gfCNCPoint6[9679] = {X 429.6854, Y 18.4377, Z -8.0000, A 0.000, B 0.000, C 0.000 }
gfCNCPoint6[9680] = {X 430.1103, Y 16.6184, Z -8.0000, A 0.000, B 0.000, C 0.000 }
gfCNCPoint6[9681] = {X 430.6685, Y 15.1182, Z -8.0000, A 0.000, B 0.000, C 0.000 }
gfCNCPoint6[9682] = {X 431.4282, Y 13.7093, Z -8.0000, A 0.000, B 0.000, C 0.000 }
gfCNCPoint6[9683] = {X 432.3747, Y 12.4184, Z -8.0000, A 0.000, B 0.000, C 0.000 }
gfCNCPoint6[9684] = {X 433.4901, Y 11.2703, Z -8.0000, A 0.000, B 0.000, C 0.000 }
gfCNCPoint6[9685] = {X 434.7530, Y 10.2868, Z -8.0000, A 0.000, B 0.000, C 0.000 }
gfCNCPoint6[9686] = {X 436.1394, Y 9.4867, Z -8.0000, A 0.000, B 0.000, C 0.000 }
gfCNCPoint6[9687] = {X 437.6228, Y 8.8852, Z -8.0000, A 0.000, B 0.000, C 0.000 }
gfCNCPoint6[9688] = {X 439.1749, Y 8.4939, Z -8.0000, A 0.000, B 0.000, C 0.000 }
gfCNCPoint6[9689] = {X 441.2506, Y 8.2065, Z -8.0000, A 0.000, B 0.000, C 0.000 }
gfCNCPoint6[9690] = {X 443.3440, Y 8.1133, Z -8.0000, A 0.000, B 0.000, C 0.000 }
gfCNCPoint6[9691] = {X 444.0364, Y 8.1092, Z -8.0000, A 0.000, B 0.000, C 0.000 }
gfCNCPoint6[9692] = {X 459.4469, Y 8.1092, Z -8.0000, A 0.000, B 0.000, C 0.000 }
gfCNCPoint6[9693] = {X 460.3528, Y 8.2113, Z -8.0000, A 0.000, B 0.000, C 0.000 }
gfCNCPoint6[9694] = {X 461.2133, Y 8.5124, Z -8.0000, A 0.000, B 0.000, C 0.000 }
gfCNCPoint6[9695] = {X 461.9852, Y 8.9974, Z -8.0000, A 0.000, B 0.000, C 0.000 }
gfCNCPoint6[9696] = {X 462.6298, Y 9.6420, Z -8.0000, A 0.000, B 0.000, C 0.000 }
gfCNCPoint6[9697] = {X 463.1148, Y 10.4139, Z -8.0000, A 0.000, B 0.000, C 0.000 }
gfCNCPoint6[9698] = {X 463.4159, Y 11.2744, Z -8.0000, A 0.000, B 0.000, C 0.000 }
gfCNCPoint6[9699] = {X 463.5179, Y 12.1803, Z -8.0000, A 0.000, B 0.000, C 0.000 }
gfCNCPoint6[9700] = {X 463.5179, Y 12.9782, Z -8.0000, A 0.000, B 0.000, C 0.000 }
gfCNCPoint6[9701] = {X 463.4242, Y 13.8477, Z -8.0000, A 0.000, B 0.000, C 0.000 }
gfCNCPoint6[9702] = {X 463.1473, Y 14.6772, Z -8.0000, A 0.000, B 0.000, C 0.000 }
gfCNCPoint6[9703] = {X 462.6999, Y 15.4287, Z -8.0000, A 0.000, B 0.000, C 0.000 }
gfCNCPoint6[9704] = {X 462.1027, Y 16.0676, Z -8.0000, A 0.000, B 0.000, C 0.000 }
gfCNCPoint6[9705] = {X 462.0451, Y 16.1164, Z -8.0000, A 0.000, B 0.000, C 0.000 }
gfCNCPoint6[9706] = {X 461.9865, Y 16.1641, Z -8.0000, A 0.000, B 0.000, C 0.000 }
gfCNCPoint6[9707] = {X 461.9918, Y 16.1980, Z -8.0000, A 0.000, B 0.000, C 0.000 }
gfCNCPoint6[9708] = {X 461.9920, Y 28.5935, Z -8.0000, A 0.000, B 0.000, C 0.000 }
gfCNCPoint6[9709] = {X 465.9920, Y 28.5934, Z -8.0000, A 0.000, B 0.000, C 0.000 }
gfCNCPoint6[9710] = {X 465.9920, Y 28.5933, Z -8.0000, A 0.000, B 0.000, C 0.000 }
gfCNCPoint6[9711] = {X 461.9118, Y 28.5935, Z -8.0000, A 0.000, B 0.000, C 0.000 }
gfCNCPoint6[9712] = {X 461.9123, Y 41.0648, Z -8.0000, A 0.000, B 0.000, C 0.000 }
gfCNCPoint6[9713] = {X 462.0510, Y 41.1802, Z -8.0000, A 0.000, B 0.000, C 0.000 }
gfCNCPoint6[9714] = {X 462.6363, Y 41.8066, Z -8.0000, A 0.000, B 0.000, C 0.000 }
gfCNCPoint6[9715] = {X 463.0747, Y 42.5433, Z -8.0000, A 0.000, B 0.000, C 0.000 }
gfCNCPoint6[9716] = {X 463.3461, Y 43.3565, Z -8.0000, A 0.000, B 0.000, C 0.000 }
gfCNCPoint6[9717] = {X 463.4379, Y 44.2088, Z -8.0000, A 0.000, B 0.000, C 0.000 }
gfCNCPoint6[9718] = {X 463.4379, Y 45.0000, Z -8.0000, A 0.000, B 0.000, C 0.000 }
gfCNCPoint6[9719] = {X 463.3377, Y 45.8901, Z -8.0000, A 0.000, B 0.000, C 0.000 }
gfCNCPoint6[9720] = {X 463.0418, Y 46.7355, Z -8.0000, A 0.000, B 0.000, C 0.000 }
gfCNCPoint6[9721] = {X 462.5653, Y 47.4940, Z -8.0000, A 0.000, B 0.000, C 0.000 }
gfCNCPoint6[9722] = {X 461.9319, Y 48.1273, Z -8.0000, A 0.000, B 0.000, C 0.000 }
gfCNCPoint6[9723] = {X 461.1735, Y 48.6039, Z -8.0000, A 0.000, B 0.000, C 0.000 }
gfCNCPoint6[9724] = {X 460.3280, Y 48.8997, Z -8.0000, A 0.000, B 0.000, C 0.000 }
gfCNCPoint6[9725] = {X 459.4379, Y 49.0000, Z -8.0000, A 0.000, B 0.000, C 0.000 }
gfCNCPoint6[9726] = {X 452.9945, Y 49.0000, Z -8.0000, A 0.000, B 0.000, C 0.000 }
gfCNCPoint6[9727] = {X 452.1044, Y 48.8997, Z -8.0000, A 0.000, B 0.000, C 0.000 }
gfCNCPoint6[9728] = {X 451.2589, Y 48.6039, Z -8.0000, A 0.000, B 0.000, C 0.000 }
gfCNCPoint6[9729] = {X 450.5005, Y 48.1273, Z -8.0000, A 0.000, B 0.000, C 0.000 }
gfCNCPoint6[9730] = {X 449.8671, Y 47.4939, Z -8.0000, A 0.000, B 0.000, C 0.000 }
gfCNCPoint6[9731] = {X 449.3906, Y 46.7355, Z -8.0000, A 0.000, B 0.000, C 0.000 }
gfCNCPoint6[9732] = {X 449.0948, Y 45.8901, Z -8.0000, A 0.000, B 0.000, C 0.000 }
gfCNCPoint6[9733] = {X 448.9945, Y 45.0000, Z -8.0000, A 0.000, B 0.000, C 0.000 }
gfCNCPoint6[9734] = {X 448.9949, Y 44.1538, Z -8.0000, A 0.000, B 0.000, C 0.000 }
gfCNCPoint6[9735] = {X 449.1055, Y 43.2730, Z -8.0000, A 0.000, B 0.000, C 0.000 }
gfCNCPoint6[9736] = {X 449.4077, Y 42.4382, Z -8.0000, A 0.000, B 0.000, C 0.000 }
gfCNCPoint6[9737] = {X 449.8865, Y 41.6907, Z -8.0000, A 0.000, B 0.000, C 0.000 }
gfCNCPoint6[9738] = {X 450.5184, Y 41.0672, Z -8.0000, A 0.000, B 0.000, C 0.000 }
gfCNCPoint6[9739] = {X 450.5184, Y 34.1538, Z -8.0000, A 0.000, B 0.000, C 0.000 }
gfCNCPoint6[9740] = {X 447.2803, Y 34.1538, Z -8.0000, A 0.000, B 0.000, C 0.000 }
gfCNCPoint6[9741] = {X 442.8423, Y 42.7952, Z -8.0000, A 0.000, B 0.000, C 0.000 }
gfCNCPoint6[9742] = {X 442.8973, Y 42.9503, Z -8.0000, A 0.000, B 0.000, C 0.000 }
gfCNCPoint6[9743] = {X 443.0494, Y 43.5714, Z -8.0000, A 0.000, B 0.000, C 0.000 }
gfCNCPoint6[9744] = {X 443.1005, Y 44.2089, Z -8.0000, A 0.000, B 0.000, C 0.000 }
gfCNCPoint6[9745] = {X 443.1005, Y 45.0000, Z -8.0000, A 0.000, B 0.000, C 0.000 }
gfCNCPoint6[9746] = {X 443.0002, Y 45.8901, Z -8.0000, A 0.000, B 0.000, C 0.000 }
gfCNCPoint6[9747] = {X 442.7043, Y 46.7355, Z -8.0000, A 0.000, B 0.000, C 0.000 }
gfCNCPoint6[9748] = {X 442.2278, Y 47.4940, Z -8.0000, A 0.000, B 0.000, C 0.000 }
gfCNCPoint6[9749] = {X 441.5944, Y 48.1273, Z -8.0000, A 0.000, B 0.000, C 0.000 }
gfCNCPoint6[9750] = {X 440.8360, Y 48.6039, Z -8.0000, A 0.000, B 0.000, C 0.000 }
gfCNCPoint6[9751] = {X 439.9906, Y 48.8997, Z -8.0000, A 0.000, B 0.000, C 0.000 }
gfCNCPoint6[9752] = {X 439.1005, Y 49.0000, Z -8.0000, A 0.000, B 0.000, C 0.000 }
gfCNCPoint6[9753] = {X 432.5144, Y 49.0000, Z -8.0000, A 0.000, B 0.000, C 0.000 }
gfCNCPoint6[9754] = {X 431.6243, Y 48.8997, Z -8.0000, A 0.000, B 0.000, C 0.000 }
gfCNCPoint6[9755] = {X 430.7789, Y 48.6039, Z -8.0000, A 0.000, B 0.000, C 0.000 }
gfCNCPoint6[9756] = {X 430.0204, Y 48.1273, Z -8.0000, A 0.000, B 0.000, C 0.000 }
gfCNCPoint6[9757] = {X 429.3871, Y 47.4940, Z -8.0000, A 0.000, B 0.000, C 0.000 }
gfCNCPoint6[9758] = {X 428.9105, Y 46.7355, Z -8.0000, A 0.000, B 0.000, C 0.000 }
gfCNCPoint6[9759] = {X 428.6147, Y 45.8901, Z -8.0000, A 0.000, B 0.000, C 0.000 }
gfCNCPoint6[9760] = {X 428.5144, Y 45.0000, Z -8.0000, A 0.000, B 0.000, C 0.000 }
gfCNCPoint6[9761] = {X 428.5148, Y 44.1538, Z -8.0000, A 0.000, B 0.000, C 0.000 }
gfCNCPoint6[9762] = {X 428.6096, Y 43.3414, Z -8.0000, A 0.000, B 0.000, C 0.000 }
gfCNCPoint6[9763] = {X 428.8676, Y 42.5654, Z -8.0000, A 0.000, B 0.000, C 0.000 }
gfCNCPoint6[9764] = {X 429.2781, Y 41.8580, Z -8.0000, A 0.000, B 0.000, C 0.000 }
gfCNCPoint6[9765] = {X 429.8239, Y 41.2489, Z -8.0000, A 0.000, B 0.000, C 0.000 }
gfCNCPoint6[9766] = {X 430.4821, Y 40.7635, Z -8.0000, A 0.000, B 0.000, C 0.000 }
gfCNCPoint6[9767] = {X 431.2253, Y 40.4222, Z -8.0000, A 0.000, B 0.000, C 0.000 }
gfCNCPoint6[9768] = {X 435.4110, Y 32.2292, Z -8.0000, A 0.000, B 0.000, C 0.000 }
gfCNCPoint6[9769] = {X 434.2190, Y 31.4711, Z -8.0000, A 0.000, B 0.000, C 0.000 }
gfCNCPoint6[9770] = {X 433.1339, Y 30.5665, Z -8.0000, A 0.000, B 0.000, C 0.000 }
gfCNCPoint6[9771] = {X 432.1736, Y 29.5306, Z -8.0000, A 0.000, B 0.000, C 0.000 }
gfCNCPoint6[9772] = {X 431.3537, Y 28.3802, Z -8.0000, A 0.000, B 0.000, C 0.000 }
gfCNCPoint6[9773] = {X 430.6879, Y 27.1343, Z -8.0000, A 0.000, B 0.000, C 0.000 }
gfCNCPoint6[9774] = {X 430.1870, Y 25.8134, Z -8.0000, A 0.000, B 0.000, C 0.000 }
gfCNCPoint6[9775] = {X 429.7643, Y 24.0033, Z -8.0000, A 0.000, B 0.000, C 0.000 }
gfCNCPoint6[9776] = {X 429.5515, Y 22.1566, Z -8.0000, A 0.000, B 0.000, C 0.000 }
gfCNCPoint6[9777] = {X 429.5515, Y 20.2978, Z -8.0000, A 0.000, B 0.000, C 0.000 }
gfCNCPoint6[9778] = {X 429.7643, Y 18.4512, Z -8.0000, A 0.000, B 0.000, C 0.000 }
gfCNCPoint6[9779] = {X 430.1870, Y 16.6411, Z -8.0000, A 0.000, B 0.000, C 0.000 }
gfCNCPoint6[9780] = {X 430.7414, Y 15.1512, Z -8.0000, A 0.000, B 0.000, C 0.000 }
gfCNCPoint6[9781] = {X 431.4958, Y 13.7519, Z -8.0000, A 0.000, B 0.000, C 0.000 }
gfCNCPoint6[9782] = {X 432.4359, Y 12.4700, Z -8.0000, A 0.000, B 0.000, C 0.000 }
gfCNCPoint6[9783] = {X 433.5436, Y 11.3298, Z -8.0000, A 0.000, B 0.000, C 0.000 }
gfCNCPoint6[9784] = {X 434.7978, Y 10.3531, Z -8.0000, A 0.000, B 0.000, C 0.000 }
gfCNCPoint6[9785] = {X 436.1746, Y 9.5585, Z -8.0000, A 0.000, B 0.000, C 0.000 }
gfCNCPoint6[9786] = {X 437.6478, Y 8.9612, Z -8.0000, A 0.000, B 0.000, C 0.000 }
gfCNCPoint6[9787] = {X 439.1893, Y 8.5726, Z -8.0000, A 0.000, B 0.000, C 0.000 }
gfCNCPoint6[9788] = {X 441.2579, Y 8.2861, Z -8.0000, A 0.000, B 0.000, C 0.000 }
gfCNCPoint6[9789] = {X 443.3442, Y 8.1933, Z -8.0000, A 0.000, B 0.000, C 0.000 }
gfCNCPoint6[9790] = {X 444.0367, Y 8.1892, Z -8.0000, A 0.000, B 0.000, C 0.000 }
gfCNCPoint6[9791] = {X 459.4469, Y 8.1892, Z -8.0000, A 0.000, B 0.000, C 0.000 }
gfCNCPoint6[9792] = {X 460.3350, Y 8.2893, Z -8.0000, A 0.000, B 0.000, C 0.000 }
gfCNCPoint6[9793] = {X 461.1786, Y 8.5845, Z -8.0000, A 0.000, B 0.000, C 0.000 }
gfCNCPoint6[9794] = {X 461.9353, Y 9.0600, Z -8.0000, A 0.000, B 0.000, C 0.000 }
gfCNCPoint6[9795] = {X 462.5672, Y 9.6919, Z -8.0000, A 0.000, B 0.000, C 0.000 }
gfCNCPoint6[9796] = {X 463.0427, Y 10.4486, Z -8.0000, A 0.000, B 0.000, C 0.000 }
gfCNCPoint6[9797] = {X 463.3379, Y 11.2922, Z -8.0000, A 0.000, B 0.000, C 0.000 }
gfCNCPoint6[9798] = {X 463.4379, Y 12.1803, Z -8.0000, A 0.000, B 0.000, C 0.000 }
gfCNCPoint6[9799] = {X 463.4378, Y 13.0163, Z -8.0000, A 0.000, B 0.000, C 0.000 }
gfCNCPoint6[9800] = {X 463.3398, Y 13.8585, Z -8.0000, A 0.000, B 0.000, C 0.000 }
gfCNCPoint6[9801] = {X 463.0666, Y 14.6612, Z -8.0000, A 0.000, B 0.000, C 0.000 }
gfCNCPoint6[9802] = {X 462.6302, Y 15.3883, Z -8.0000, A 0.000, B 0.000, C 0.000 }
gfCNCPoint6[9803] = {X 462.0505, Y 16.0070, Z -8.0000, A 0.000, B 0.000, C 0.000 }
gfCNCPoint6[9804] = {X 461.9731, Y 16.0720, Z -8.0000, A 0.000, B 0.000, C 0.000 }
gfCNCPoint6[9805] = {X 461.8942, Y 16.1351, Z -8.0000, A 0.000, B 0.000, C 0.000 }
gfCNCPoint6[9806] = {X 461.9118, Y 16.1935, Z -8.0000, A 0.000, B 0.000, C 0.000 }
gfCNCPoint6[9807] = {X 461.9113, Y 16.7687, Z -8.0000, A 0.000, B 0.000, C 0.000 }
gfCNCPoint6[9808] = {X 461.9118, Y 28.5935, Z -8.0000, A 0.000, B 0.000, C 0.000 }
gfCNCPoint6[9809] = {X 465.9920, Y 28.5933, Z -8.0000, A 0.000, B 0.000, C 0.000 }
gfCNCPoint6[9810] = {X 465.9920, Y 28.5933, Z -5.0000, A 0.000, B 0.000, C 0.000 }
gfCNCPoint6[9811] = {X 465.9920, Y 28.5933, Z 11.0000, A 0.000, B 0.000, C 0.000 }
gfCNCPoint6[9812] = {X 492.3835, Y 3.7892, Z 11.0000, A 0.000, B 0.000, C 0.000 }
gfCNCPoint6[9813] = {X 492.3835, Y 3.7892, Z -5.0000, A 0.000, B 0.000, C 0.000 }
gfCNCPoint6[9814] = {X 492.3835, Y 3.7892, Z -8.0000, A 0.000, B 0.000, C 0.000 }
gfCNCPoint6[9815] = {X 492.3835, Y 7.8692, Z -8.0000, A 0.000, B 0.000, C 0.000 }
gfCNCPoint6[9816] = {X 502.2066, Y 7.8692, Z -8.0000, A 0.000, B 0.000, C 0.000 }
gfCNCPoint6[9817] = {X 502.7394, Y 7.8734, Z -8.0000, A 0.000, B 0.000, C 0.000 }
gfCNCPoint6[9818] = {X 503.6913, Y 7.9876, Z -8.0000, A 0.000, B 0.000, C 0.000 }
gfCNCPoint6[9819] = {X 504.5943, Y 8.3098, Z -8.0000, A 0.000, B 0.000, C 0.000 }
gfCNCPoint6[9820] = {X 505.4035, Y 8.8240, Z -8.0000, A 0.000, B 0.000, C 0.000 }
gfCNCPoint6[9821] = {X 506.0787, Y 9.5045, Z -8.0000, A 0.000, B 0.000, C 0.000 }
gfCNCPoint6[9822] = {X 506.5865, Y 10.3177, Z -8.0000, A 0.000, B 0.000, C 0.000 }
gfCNCPoint6[9823] = {X 506.9017, Y 11.2232, Z -8.0000, A 0.000, B 0.000, C 0.000 }
gfCNCPoint6[9824] = {X 507.0085, Y 12.1759, Z -8.0000, A 0.000, B 0.000, C 0.000 }
gfCNCPoint6[9825] = {X 507.0085, Y 12.9782, Z -8.0000, A 0.000, B 0.000, C 0.000 }
gfCNCPoint6[9826] = {X 506.9072, Y 13.9079, Z -8.0000, A 0.000, B 0.000, C 0.000 }
gfCNCPoint6[9827] = {X 506.6082, Y 14.7940, Z -8.0000, A 0.000, B 0.000, C 0.000 }
gfCNCPoint6[9828] = {X 506.1256, Y 15.5951, Z -8.0000, A 0.000, B 0.000, C 0.000 }
gfCNCPoint6[9829] = {X 505.4818, Y 16.2734, Z -8.0000, A 0.000, B 0.000, C 0.000 }
gfCNCPoint6[9830] = {X 505.4824, Y 40.9138, Z -8.0000, A 0.000, B 0.000, C 0.000 }
gfCNCPoint6[9831] = {X 506.1202, Y 41.5848, Z -8.0000, A 0.000, B 0.000, C 0.000 }
gfCNCPoint6[9832] = {X 506.6005, Y 42.3762, Z -8.0000, A 0.000, B 0.000, C 0.000 }
gfCNCPoint6[9833] = {X 506.9012, Y 43.2518, Z -8.0000, A 0.000, B 0.000, C 0.000 }
gfCNCPoint6[9834] = {X 507.0083, Y 44.1713, Z -8.0000, A 0.000, B 0.000, C 0.000 }
gfCNCPoint6[9835] = {X 507.0085, Y 45.0000, Z -8.0000, A 0.000, B 0.000, C 0.000 }
gfCNCPoint6[9836] = {X 506.9002, Y 45.9613, Z -8.0000, A 0.000, B 0.000, C 0.000 }
gfCNCPoint6[9837] = {X 506.5807, Y 46.8744, Z -8.0000, A 0.000, B 0.000, C 0.000 }
gfCNCPoint6[9838] = {X 506.0660, Y 47.6935, Z -8.0000, A 0.000, B 0.000, C 0.000 }
gfCNCPoint6[9839] = {X 505.3820, Y 48.3775, Z -8.0000, A 0.000, B 0.000, C 0.000 }
gfCNCPoint6[9840] = {X 504.5629, Y 48.8922, Z -8.0000, A 0.000, B 0.000, C 0.000 }
gfCNCPoint6[9841] = {X 503.6498, Y 49.2117, Z -8.0000, A 0.000, B 0.000, C 0.000 }
gfCNCPoint6[9842] = {X 502.6885, Y 49.3200, Z -8.0000, A 0.000, B 0.000, C 0.000 }
gfCNCPoint6[9843] = {X 496.2450, Y 49.3200, Z -8.0000, A 0.000, B 0.000, C 0.000 }
gfCNCPoint6[9844] = {X 495.2885, Y 49.2128, Z -8.0000, A 0.000, B 0.000, C 0.000 }
gfCNCPoint6[9845] = {X 494.3794, Y 48.8964, Z -8.0000, A 0.000, B 0.000, C 0.000 }
gfCNCPoint6[9846] = {X 493.5630, Y 48.3866, Z -8.0000, A 0.000, B 0.000, C 0.000 }
gfCNCPoint6[9847] = {X 492.8797, Y 47.7087, Z -8.0000, A 0.000, B 0.000, C 0.000 }
gfCNCPoint6[9848] = {X 492.3635, Y 46.8963, Z -8.0000, A 0.000, B 0.000, C 0.000 }
gfCNCPoint6[9849] = {X 492.0399, Y 45.9898, Z -8.0000, A 0.000, B 0.000, C 0.000 }
gfCNCPoint6[9850] = {X 491.9252, Y 45.0341, Z -8.0000, A 0.000, B 0.000, C 0.000 }
gfCNCPoint6[9851] = {X 491.9254, Y 44.1494, Z -8.0000, A 0.000, B 0.000, C 0.000 }
gfCNCPoint6[9852] = {X 492.0359, Y 43.2364, Z -8.0000, A 0.000, B 0.000, C 0.000 }
gfCNCPoint6[9853] = {X 492.3371, Y 42.3675, Z -8.0000, A 0.000, B 0.000, C 0.000 }
gfCNCPoint6[9854] = {X 492.8153, Y 41.5821, Z -8.0000, A 0.000, B 0.000, C 0.000 }
gfCNCPoint6[9855] = {X 493.4490, Y 40.9157, Z -8.0000, A 0.000, B 0.000, C 0.000 }
gfCNCPoint6[9856] = {X 493.4490, Y 34.4738, Z -8.0000, A 0.000, B 0.000, C 0.000 }
gfCNCPoint6[9857] = {X 490.7257, Y 34.4738, Z -8.0000, A 0.000, B 0.000, C 0.000 }
gfCNCPoint6[9858] = {X 486.4408, Y 42.8183, Z -8.0000, A 0.000, B 0.000, C 0.000 }
gfCNCPoint6[9859] = {X 486.4455, Y 42.8311, Z -8.0000, A 0.000, B 0.000, C 0.000 }
gfCNCPoint6[9860] = {X 486.6111, Y 43.4916, Z -8.0000, A 0.000, B 0.000, C 0.000 }
gfCNCPoint6[9861] = {X 486.6708, Y 44.1699, Z -8.0000, A 0.000, B 0.000, C 0.000 }
gfCNCPoint6[9862] = {X 486.6710, Y 45.0000, Z -8.0000, A 0.000, B 0.000, C 0.000 }
gfCNCPoint6[9863] = {X 486.5627, Y 45.9613, Z -8.0000, A 0.000, B 0.000, C 0.000 }
gfCNCPoint6[9864] = {X 486.2432, Y 46.8744, Z -8.0000, A 0.000, B 0.000, C 0.000 }
gfCNCPoint6[9865] = {X 485.7285, Y 47.6935, Z -8.0000, A 0.000, B 0.000, C 0.000 }
gfCNCPoint6[9866] = {X 485.0445, Y 48.3775, Z -8.0000, A 0.000, B 0.000, C 0.000 }
gfCNCPoint6[9867] = {X 484.2254, Y 48.8922, Z -8.0000, A 0.000, B 0.000, C 0.000 }
gfCNCPoint6[9868] = {X 483.3123, Y 49.2117, Z -8.0000, A 0.000, B 0.000, C 0.000 }
gfCNCPoint6[9869] = {X 482.3510, Y 49.3200, Z -8.0000, A 0.000, B 0.000, C 0.000 }
gfCNCPoint6[9870] = {X 475.7650, Y 49.3200, Z -8.0000, A 0.000, B 0.000, C 0.000 }
gfCNCPoint6[9871] = {X 474.8037, Y 49.2117, Z -8.0000, A 0.000, B 0.000, C 0.000 }
gfCNCPoint6[9872] = {X 473.8906, Y 48.8922, Z -8.0000, A 0.000, B 0.000, C 0.000 }
gfCNCPoint6[9873] = {X 473.0715, Y 48.3775, Z -8.0000, A 0.000, B 0.000, C 0.000 }
gfCNCPoint6[9874] = {X 472.3875, Y 47.6935, Z -8.0000, A 0.000, B 0.000, C 0.000 }
gfCNCPoint6[9875] = {X 471.8728, Y 46.8745, Z -8.0000, A 0.000, B 0.000, C 0.000 }
gfCNCPoint6[9876] = {X 471.5533, Y 45.9614, Z -8.0000, A 0.000, B 0.000, C 0.000 }
gfCNCPoint6[9877] = {X 471.4450, Y 45.0001, Z -8.0000, A 0.000, B 0.000, C 0.000 }
gfCNCPoint6[9878] = {X 471.4454, Y 44.1494, Z -8.0000, A 0.000, B 0.000, C 0.000 }
gfCNCPoint6[9879] = {X 471.5430, Y 43.2935, Z -8.0000, A 0.000, B 0.000, C 0.000 }
gfCNCPoint6[9880] = {X 471.8086, Y 42.4740, Z -8.0000, A 0.000, B 0.000, C 0.000 }
gfCNCPoint6[9881] = {X 472.2314, Y 41.7236, Z -8.0000, A 0.000, B 0.000, C 0.000 }
gfCNCPoint6[9882] = {X 472.7947, Y 41.0719, Z -8.0000, A 0.000, B 0.000, C 0.000 }
gfCNCPoint6[9883] = {X 473.4762, Y 40.5449, Z -8.0000, A 0.000, B 0.000, C 0.000 }
gfCNCPoint6[9884] = {X 474.2486, Y 40.1637, Z -8.0000, A 0.000, B 0.000, C 0.000 }
gfCNCPoint6[9885] = {X 478.2329, Y 32.3647, Z -8.0000, A 0.000, B 0.000, C 0.000 }
gfCNCPoint6[9886] = {X 476.9687, Y 31.4977, Z -8.0000, A 0.000, B 0.000, C 0.000 }
gfCNCPoint6[9887] = {X 475.8315, Y 30.4696, Z -8.0000, A 0.000, B 0.000, C 0.000 }
gfCNCPoint6[9888] = {X 474.8419, Y 29.2989, Z -8.0000, A 0.000, B 0.000, C 0.000 }
gfCNCPoint6[9889] = {X 474.0174, Y 28.0065, Z -8.0000, A 0.000, B 0.000, C 0.000 }
gfCNCPoint6[9890] = {X 473.3730, Y 26.6155, Z -8.0000, A 0.000, B 0.000, C 0.000 }
gfCNCPoint6[9891] = {X 472.9201, Y 25.1510, Z -8.0000, A 0.000, B 0.000, C 0.000 }
gfCNCPoint6[9892] = {X 472.6065, Y 23.4679, Z -8.0000, A 0.000, B 0.000, C 0.000 }
gfCNCPoint6[9893] = {X 472.4664, Y 21.7615, Z -8.0000, A 0.000, B 0.000, C 0.000 }
gfCNCPoint6[9894] = {X 472.5011, Y 20.0498, Z -8.0000, A 0.000, B 0.000, C 0.000 }
gfCNCPoint6[9895] = {X 472.7103, Y 18.3506, Z -8.0000, A 0.000, B 0.000, C 0.000 }
gfCNCPoint6[9896] = {X 473.0918, Y 16.6816, Z -8.0000, A 0.000, B 0.000, C 0.000 }
gfCNCPoint6[9897] = {X 473.6348, Y 15.1666, Z -8.0000, A 0.000, B 0.000, C 0.000 }
gfCNCPoint6[9898] = {X 474.3784, Y 13.7393, Z -8.0000, A 0.000, B 0.000, C 0.000 }
gfCNCPoint6[9899] = {X 475.3086, Y 12.4261, Z -8.0000, A 0.000, B 0.000, C 0.000 }
gfCNCPoint6[9900] = {X 476.4085, Y 11.2512, Z -8.0000, A 0.000, B 0.000, C 0.000 }
gfCNCPoint6[9901] = {X 477.6575, Y 10.2363, Z -8.0000, A 0.000, B 0.000, C 0.000 }
gfCNCPoint6[9902] = {X 479.0327, Y 9.4003, Z -8.0000, A 0.000, B 0.000, C 0.000 }
gfCNCPoint6[9903] = {X 480.5085, Y 8.7585, Z -8.0000, A 0.000, B 0.000, C 0.000 }
gfCNCPoint6[9904] = {X 482.0578, Y 8.3229, Z -8.0000, A 0.000, B 0.000, C 0.000 }
gfCNCPoint6[9905] = {X 484.1552, Y 7.9961, Z -8.0000, A 0.000, B 0.000, C 0.000 }
gfCNCPoint6[9906] = {X 486.2747, Y 7.8814, Z -8.0000, A 0.000, B 0.000, C 0.000 }
gfCNCPoint6[9907] = {X 486.9679, Y 7.8692, Z -8.0000, A 0.000, B 0.000, C 0.000 }
gfCNCPoint6[9908] = {X 492.3835, Y 7.8692, Z -8.0000, A 0.000, B 0.000, C 0.000 }
gfCNCPoint6[9909] = {X 492.3835, Y 3.8692, Z -8.0000, A 0.000, B 0.000, C 0.000 }
gfCNCPoint6[9910] = {X 492.3835, Y 7.9492, Z -8.0000, A 0.000, B 0.000, C 0.000 }
gfCNCPoint6[9911] = {X 502.2063, Y 7.9492, Z -8.0000, A 0.000, B 0.000, C 0.000 }
gfCNCPoint6[9912] = {X 502.7388, Y 7.9534, Z -8.0000, A 0.000, B 0.000, C 0.000 }
gfCNCPoint6[9913] = {X 503.6730, Y 8.0655, Z -8.0000, A 0.000, B 0.000, C 0.000 }
gfCNCPoint6[9914] = {X 504.5592, Y 8.3817, Z -8.0000, A 0.000, B 0.000, C 0.000 }
gfCNCPoint6[9915] = {X 505.3533, Y 8.8863, Z -8.0000, A 0.000, B 0.000, C 0.000 }
gfCNCPoint6[9916] = {X 506.0160, Y 9.5542, Z -8.0000, A 0.000, B 0.000, C 0.000 }
gfCNCPoint6[9917] = {X 506.5144, Y 10.3523, Z -8.0000, A 0.000, B 0.000, C 0.000 }
gfCNCPoint6[9918] = {X 506.8237, Y 11.2409, Z -8.0000, A 0.000, B 0.000, C 0.000 }
gfCNCPoint6[9919] = {X 506.9285, Y 12.1759, Z -8.0000, A 0.000, B 0.000, C 0.000 }
gfCNCPoint6[9920] = {X 506.9285, Y 12.9782, Z -8.0000, A 0.000, B 0.000, C 0.000 }
gfCNCPoint6[9921] = {X 506.8271, Y 13.8997, Z -8.0000, A 0.000, B 0.000, C 0.000 }
gfCNCPoint6[9922] = {X 506.5279, Y 14.7771, Z -8.0000, A 0.000, B 0.000, C 0.000 }
gfCNCPoint6[9923] = {X 506.0451, Y 15.5686, Z -8.0000, A 0.000, B 0.000, C 0.000 }
gfCNCPoint6[9924] = {X 505.4018, Y 16.2362, Z -8.0000, A 0.000, B 0.000, C 0.000 }
gfCNCPoint6[9925] = {X 505.4024, Y 40.9514, Z -8.0000, A 0.000, B 0.000, C 0.000 }
gfCNCPoint6[9926] = {X 505.4306, Y 40.9749, Z -8.0000, A 0.000, B 0.000, C 0.000 }
gfCNCPoint6[9927] = {X 506.0567, Y 41.6334, Z -8.0000, A 0.000, B 0.000, C 0.000 }
gfCNCPoint6[9928] = {X 506.5281, Y 42.4101, Z -8.0000, A 0.000, B 0.000, C 0.000 }
gfCNCPoint6[9929] = {X 506.8231, Y 43.2695, Z -8.0000, A 0.000, B 0.000, C 0.000 }
gfCNCPoint6[9930] = {X 506.9283, Y 44.1720, Z -8.0000, A 0.000, B 0.000, C 0.000 }
gfCNCPoint6[9931] = {X 506.9285, Y 45.0000, Z -8.0000, A 0.000, B 0.000, C 0.000 }
gfCNCPoint6[9932] = {X 506.8222, Y 45.9435, Z -8.0000, A 0.000, B 0.000, C 0.000 }
gfCNCPoint6[9933] = {X 506.5086, Y 46.8397, Z -8.0000, A 0.000, B 0.000, C 0.000 }
gfCNCPoint6[9934] = {X 506.0035, Y 47.6436, Z -8.0000, A 0.000, B 0.000, C 0.000 }
gfCNCPoint6[9935] = {X 505.3321, Y 48.3150, Z -8.0000, A 0.000, B 0.000, C 0.000 }
gfCNCPoint6[9936] = {X 504.5282, Y 48.8201, Z -8.0000, A 0.000, B 0.000, C 0.000 }
gfCNCPoint6[9937] = {X 503.6320, Y 49.1337, Z -8.0000, A 0.000, B 0.000, C 0.000 }
gfCNCPoint6[9938] = {X 502.6885, Y 49.2400, Z -8.0000, A 0.000, B 0.000, C 0.000 }
gfCNCPoint6[9939] = {X 496.2450, Y 49.2400, Z -8.0000, A 0.000, B 0.000, C 0.000 }
gfCNCPoint6[9940] = {X 495.3062, Y 49.1348, Z -8.0000, A 0.000, B 0.000, C 0.000 }
gfCNCPoint6[9941] = {X 494.4140, Y 48.8242, Z -8.0000, A 0.000, B 0.000, C 0.000 }
gfCNCPoint6[9942] = {X 493.6127, Y 48.3239, Z -8.0000, A 0.000, B 0.000, C 0.000 }
gfCNCPoint6[9943] = {X 492.9420, Y 47.6585, Z -8.0000, A 0.000, B 0.000, C 0.000 }
gfCNCPoint6[9944] = {X 492.4354, Y 46.8612, Z -8.0000, A 0.000, B 0.000, C 0.000 }
gfCNCPoint6[9945] = {X 492.1178, Y 45.9714, Z -8.0000, A 0.000, B 0.000, C 0.000 }
gfCNCPoint6[9946] = {X 492.0052, Y 45.0335, Z -8.0000, A 0.000, B 0.000, C 0.000 }
gfCNCPoint6[9947] = {X 492.0054, Y 44.1505, Z -8.0000, A 0.000, B 0.000, C 0.000 }
gfCNCPoint6[9948] = {X 492.1159, Y 43.2454, Z -8.0000, A 0.000, B 0.000, C 0.000 }
gfCNCPoint6[9949] = {X 492.4173, Y 42.3850, Z -8.0000, A 0.000, B 0.000, C 0.000 }
gfCNCPoint6[9950] = {X 492.8957, Y 41.6088, Z -8.0000, A 0.000, B 0.000, C 0.000 }
gfCNCPoint6[9951] = {X 493.5290, Y 40.9529, Z -8.0000, A 0.000, B 0.000, C 0.000 }
gfCNCPoint6[9952] = {X 493.5290, Y 34.3938, Z -8.0000, A 0.000, B 0.000, C 0.000 }
gfCNCPoint6[9953] = {X 490.6769, Y 34.3938, Z -8.0000, A 0.000, B 0.000, C 0.000 }
gfCNCPoint6[9954] = {X 486.3536, Y 42.8129, Z -8.0000, A 0.000, B 0.000, C 0.000 }
gfCNCPoint6[9955] = {X 486.3700, Y 42.8576, Z -8.0000, A 0.000, B 0.000, C 0.000 }
gfCNCPoint6[9956] = {X 486.5323, Y 43.5054, Z -8.0000, A 0.000, B 0.000, C 0.000 }
gfCNCPoint6[9957] = {X 486.5908, Y 44.1706, Z -8.0000, A 0.000, B 0.000, C 0.000 }
gfCNCPoint6[9958] = {X 486.5910, Y 45.0000, Z -8.0000, A 0.000, B 0.000, C 0.000 }
gfCNCPoint6[9959] = {X 486.4847, Y 45.9435, Z -8.0000, A 0.000, B 0.000, C 0.000 }
gfCNCPoint6[9960] = {X 486.1711, Y 46.8397, Z -8.0000, A 0.000, B 0.000, C 0.000 }
gfCNCPoint6[9961] = {X 485.6660, Y 47.6436, Z -8.0000, A 0.000, B 0.000, C 0.000 }
gfCNCPoint6[9962] = {X 484.9946, Y 48.3150, Z -8.0000, A 0.000, B 0.000, C 0.000 }
gfCNCPoint6[9963] = {X 484.1907, Y 48.8201, Z -8.0000, A 0.000, B 0.000, C 0.000 }
gfCNCPoint6[9964] = {X 483.2945, Y 49.1337, Z -8.0000, A 0.000, B 0.000, C 0.000 }
gfCNCPoint6[9965] = {X 482.3510, Y 49.2400, Z -8.0000, A 0.000, B 0.000, C 0.000 }
gfCNCPoint6[9966] = {X 475.7650, Y 49.2400, Z -8.0000, A 0.000, B 0.000, C 0.000 }
gfCNCPoint6[9967] = {X 474.8215, Y 49.1337, Z -8.0000, A 0.000, B 0.000, C 0.000 }
gfCNCPoint6[9968] = {X 473.9253, Y 48.8201, Z -8.0000, A 0.000, B 0.000, C 0.000 }
gfCNCPoint6[9969] = {X 473.1214, Y 48.3150, Z -8.0000, A 0.000, B 0.000, C 0.000 }
gfCNCPoint6[9970] = {X 472.4500, Y 47.6436, Z -8.0000, A 0.000, B 0.000, C 0.000 }
gfCNCPoint6[9971] = {X 471.9449, Y 46.8397, Z -8.0000, A 0.000, B 0.000, C 0.000 }
gfCNCPoint6[9972] = {X 471.6313, Y 45.9436, Z -8.0000, A 0.000, B 0.000, C 0.000 }
gfCNCPoint6[9973] = {X 471.5250, Y 45.0001, Z -8.0000, A 0.000, B 0.000, C 0.000 }
gfCNCPoint6[9974] = {X 471.5254, Y 44.1505, Z -8.0000, A 0.000, B 0.000, C 0.000 }
gfCNCPoint6[9975] = {X 471.6223, Y 43.3054, Z -8.0000, A 0.000, B 0.000, C 0.000 }
gfCNCPoint6[9976] = {X 471.8860, Y 42.4967, Z -8.0000, A 0.000, B 0.000, C 0.000 }
gfCNCPoint6[9977] = {X 472.3057, Y 41.7570, Z -8.0000, A 0.000, B 0.000, C 0.000 }
gfCNCPoint6[9978] = {X 472.8647, Y 41.1158, Z -8.0000, A 0.000, B 0.000, C 0.000 }
gfCNCPoint6[9979] = {X 473.5404, Y 40.5992, Z -8.0000, A 0.000, B 0.000, C 0.000 }
gfCNCPoint6[9980] = {X 474.3057, Y 40.2278, Z -8.0000, A 0.000, B 0.000, C 0.000 }
gfCNCPoint6[9981] = {X 478.3385, Y 32.3340, Z -8.0000, A 0.000, B 0.000, C 0.000 }
gfCNCPoint6[9982] = {X 477.0675, Y 31.4736, Z -8.0000, A 0.000, B 0.000, C 0.000 }
gfCNCPoint6[9983] = {X 475.9239, Y 30.4499, Z -8.0000, A 0.000, B 0.000, C 0.000 }
gfCNCPoint6[9984] = {X 474.9286, Y 29.2816, Z -8.0000, A 0.000, B 0.000, C 0.000 }
gfCNCPoint6[9985] = {X 474.0996, Y 27.9900, Z -8.0000, A 0.000, B 0.000, C 0.000 }
gfCNCPoint6[9986] = {X 473.4521, Y 26.5984, Z -8.0000, A 0.000, B 0.000, C 0.000 }
gfCNCPoint6[9987] = {X 472.9979, Y 25.1324, Z -8.0000, A 0.000, B 0.000, C 0.000 }
gfCNCPoint6[9988] = {X 472.6858, Y 23.4573, Z -8.0000, A 0.000, B 0.000, C 0.000 }
gfCNCPoint6[9989] = {X 472.5464, Y 21.7591, Z -8.0000, A 0.000, B 0.000, C 0.000 }
gfCNCPoint6[9990] = {X 472.5809, Y 20.0556, Z -8.0000, A 0.000, B 0.000, C 0.000 }
gfCNCPoint6[9991] = {X 472.7891, Y 18.3644, Z -8.0000, A 0.000, B 0.000, C 0.000 }
gfCNCPoint6[9992] = {X 473.1688, Y 16.7034, Z -8.0000, A 0.000, B 0.000, C 0.000 }
gfCNCPoint6[9993] = {X 473.7081, Y 15.1986, Z -8.0000, A 0.000, B 0.000, C 0.000 }
gfCNCPoint6[9994] = {X 474.4466, Y 13.7810, Z -8.0000, A 0.000, B 0.000, C 0.000 }
gfCNCPoint6[9995] = {X 475.3706, Y 12.4766, Z -8.0000, A 0.000, B 0.000, C 0.000 }
gfCNCPoint6[9996] = {X 476.4630, Y 11.3097, Z -8.0000, A 0.000, B 0.000, C 0.000 }
gfCNCPoint6[9997] = {X 477.7036, Y 10.3017, Z -8.0000, A 0.000, B 0.000, C 0.000 }
gfCNCPoint6[9998] = {X 479.0695, Y 9.4713, Z -8.0000, A 0.000, B 0.000, C 0.000 }
gfCNCPoint6[9999] = {X 480.5354, Y 8.8339, Z -8.0000, A 0.000, B 0.000, C 0.000 }
gfCNCPoint6[10000] = {X 482.0742, Y 8.4012, Z -8.0000, A 0.000, B 0.000, C 0.000 }
gfCNCPoint6[10001] = {X 484.1638, Y 8.0756, Z -8.0000, A 0.000, B 0.000, C 0.000 }
gfCNCPoint6[10002] = {X 486.2756, Y 7.9614, Z -8.0000, A 0.000, B 0.000, C 0.000 }
gfCNCPoint6[10003] = {X 486.9686, Y 7.9492, Z -8.0000, A 0.000, B 0.000, C 0.000 }
gfCNCPoint6[10004] = {X 492.3835, Y 7.9492, Z -8.0000, A 0.000, B 0.000, C 0.000 }
gfCNCPoint6[10005] = {X 492.3835, Y 3.9492, Z -8.0000, A 0.000, B 0.000, C 0.000 }
gfCNCPoint6[10006] = {X 492.3835, Y 8.0292, Z -8.0000, A 0.000, B 0.000, C 0.000 }
gfCNCPoint6[10007] = {X 502.2059, Y 8.0292, Z -8.0000, A 0.000, B 0.000, C 0.000 }
gfCNCPoint6[10008] = {X 502.7382, Y 8.0334, Z -8.0000, A 0.000, B 0.000, C 0.000 }
gfCNCPoint6[10009] = {X 503.6547, Y 8.1434, Z -8.0000, A 0.000, B 0.000, C 0.000 }
gfCNCPoint6[10010] = {X 504.5241, Y 8.4536, Z -8.0000, A 0.000, B 0.000, C 0.000 }
gfCNCPoint6[10011] = {X 505.3032, Y 8.9486, Z -8.0000, A 0.000, B 0.000, C 0.000 }
gfCNCPoint6[10012] = {X 505.9533, Y 9.6039, Z -8.0000, A 0.000, B 0.000, C 0.000 }
gfCNCPoint6[10013] = {X 506.4422, Y 10.3868, Z -8.0000, A 0.000, B 0.000, C 0.000 }
gfCNCPoint6[10014] = {X 506.7457, Y 11.2586, Z -8.0000, A 0.000, B 0.000, C 0.000 }
gfCNCPoint6[10015] = {X 506.8485, Y 12.1759, Z -8.0000, A 0.000, B 0.000, C 0.000 }
gfCNCPoint6[10016] = {X 506.8485, Y 12.9782, Z -8.0000, A 0.000, B 0.000, C 0.000 }
gfCNCPoint6[10017] = {X 506.7470, Y 13.8914, Z -8.0000, A 0.000, B 0.000, C 0.000 }
gfCNCPoint6[10018] = {X 506.4475, Y 14.7601, Z -8.0000, A 0.000, B 0.000, C 0.000 }
gfCNCPoint6[10019] = {X 505.9645, Y 15.5418, Z -8.0000, A 0.000, B 0.000, C 0.000 }
gfCNCPoint6[10020] = {X 505.3218, Y 16.1985, Z -8.0000, A 0.000, B 0.000, C 0.000 }
gfCNCPoint6[10021] = {X 505.3224, Y 40.9892, Z -8.0000, A 0.000, B 0.000, C 0.000 }
gfCNCPoint6[10022] = {X 505.3684, Y 41.0270, Z -8.0000, A 0.000, B 0.000, C 0.000 }
gfCNCPoint6[10023] = {X 505.9869, Y 41.6738, Z -8.0000, A 0.000, B 0.000, C 0.000 }
gfCNCPoint6[10024] = {X 506.4527, Y 42.4379, Z -8.0000, A 0.000, B 0.000, C 0.000 }
gfCNCPoint6[10025] = {X 506.7444, Y 43.2839, Z -8.0000, A 0.000, B 0.000, C 0.000 }
gfCNCPoint6[10026] = {X 506.8483, Y 44.1727, Z -8.0000, A 0.000, B 0.000, C 0.000 }
gfCNCPoint6[10027] = {X 506.8485, Y 45.0000, Z -8.0000, A 0.000, B 0.000, C 0.000 }
gfCNCPoint6[10028] = {X 506.7442, Y 45.9257, Z -8.0000, A 0.000, B 0.000, C 0.000 }
gfCNCPoint6[10029] = {X 506.4365, Y 46.8050, Z -8.0000, A 0.000, B 0.000, C 0.000 }
gfCNCPoint6[10030] = {X 505.9409, Y 47.5937, Z -8.0000, A 0.000, B 0.000, C 0.000 }
gfCNCPoint6[10031] = {X 505.2822, Y 48.2524, Z -8.0000, A 0.000, B 0.000, C 0.000 }
gfCNCPoint6[10032] = {X 504.4934, Y 48.7480, Z -8.0000, A 0.000, B 0.000, C 0.000 }
gfCNCPoint6[10033] = {X 503.6142, Y 49.0557, Z -8.0000, A 0.000, B 0.000, C 0.000 }
gfCNCPoint6[10034] = {X 502.6885, Y 49.1600, Z -8.0000, A 0.000, B 0.000, C 0.000 }
gfCNCPoint6[10035] = {X 496.2450, Y 49.1600, Z -8.0000, A 0.000, B 0.000, C 0.000 }
gfCNCPoint6[10036] = {X 495.3239, Y 49.0567, Z -8.0000, A 0.000, B 0.000, C 0.000 }
gfCNCPoint6[10037] = {X 494.4485, Y 48.7521, Z -8.0000, A 0.000, B 0.000, C 0.000 }
gfCNCPoint6[10038] = {X 493.6623, Y 48.2612, Z -8.0000, A 0.000, B 0.000, C 0.000 }
gfCNCPoint6[10039] = {X 493.0043, Y 47.6084, Z -8.0000, A 0.000, B 0.000, C 0.000 }
gfCNCPoint6[10040] = {X 492.5072, Y 46.8261, Z -8.0000, A 0.000, B 0.000, C 0.000 }
gfCNCPoint6[10041] = {X 492.1957, Y 45.9531, Z -8.0000, A 0.000, B 0.000, C 0.000 }
gfCNCPoint6[10042] = {X 492.0852, Y 45.0328, Z -8.0000, A 0.000, B 0.000, C 0.000 }
gfCNCPoint6[10043] = {X 492.0854, Y 44.1516, Z -8.0000, A 0.000, B 0.000, C 0.000 }
gfCNCPoint6[10044] = {X 492.1960, Y 43.2545, Z -8.0000, A 0.000, B 0.000, C 0.000 }
gfCNCPoint6[10045] = {X 492.4976, Y 42.4026, Z -8.0000, A 0.000, B 0.000, C 0.000 }
gfCNCPoint6[10046] = {X 492.9762, Y 41.6358, Z -8.0000, A 0.000, B 0.000, C 0.000 }
gfCNCPoint6[10047] = {X 493.6090, Y 40.9906, Z -8.0000, A 0.000, B 0.000, C 0.000 }
gfCNCPoint6[10048] = {X 493.6090, Y 34.3138, Z -8.0000, A 0.000, B 0.000, C 0.000 }
gfCNCPoint6[10049] = {X 490.6280, Y 34.3138, Z -8.0000, A 0.000, B 0.000, C 0.000 }
gfCNCPoint6[10050] = {X 486.2664, Y 42.8075, Z -8.0000, A 0.000, B 0.000, C 0.000 }
gfCNCPoint6[10051] = {X 486.2945, Y 42.8841, Z -8.0000, A 0.000, B 0.000, C 0.000 }
gfCNCPoint6[10052] = {X 486.4535, Y 43.5192, Z -8.0000, A 0.000, B 0.000, C 0.000 }
gfCNCPoint6[10053] = {X 486.5108, Y 44.1713, Z -8.0000, A 0.000, B 0.000, C 0.000 }
gfCNCPoint6[10054] = {X 486.5110, Y 45.0000, Z -8.0000, A 0.000, B 0.000, C 0.000 }
gfCNCPoint6[10055] = {X 486.4067, Y 45.9257, Z -8.0000, A 0.000, B 0.000, C 0.000 }
gfCNCPoint6[10056] = {X 486.0990, Y 46.8050, Z -8.0000, A 0.000, B 0.000, C 0.000 }
gfCNCPoint6[10057] = {X 485.6034, Y 47.5937, Z -8.0000, A 0.000, B 0.000, C 0.000 }
gfCNCPoint6[10058] = {X 484.9447, Y 48.2524, Z -8.0000, A 0.000, B 0.000, C 0.000 }
gfCNCPoint6[10059] = {X 484.1560, Y 48.7480, Z -8.0000, A 0.000, B 0.000, C 0.000 }
gfCNCPoint6[10060] = {X 483.2767, Y 49.0557, Z -8.0000, A 0.000, B 0.000, C 0.000 }
gfCNCPoint6[10061] = {X 482.3510, Y 49.1600, Z -8.0000, A 0.000, B 0.000, C 0.000 }
gfCNCPoint6[10062] = {X 475.7650, Y 49.1600, Z -8.0000, A 0.000, B 0.000, C 0.000 }
gfCNCPoint6[10063] = {X 474.8393, Y 49.0557, Z -8.0000, A 0.000, B 0.000, C 0.000 }
gfCNCPoint6[10064] = {X 473.9600, Y 48.7480, Z -8.0000, A 0.000, B 0.000, C 0.000 }
gfCNCPoint6[10065] = {X 473.1713, Y 48.2524, Z -8.0000, A 0.000, B 0.000, C 0.000 }
gfCNCPoint6[10066] = {X 472.5126, Y 47.5937, Z -8.0000, A 0.000, B 0.000, C 0.000 }
gfCNCPoint6[10067] = {X 472.0169, Y 46.8050, Z -8.0000, A 0.000, B 0.000, C 0.000 }
gfCNCPoint6[10068] = {X 471.7093, Y 45.9257, Z -8.0000, A 0.000, B 0.000, C 0.000 }
gfCNCPoint6[10069] = {X 471.6050, Y 45.0000, Z -8.0000, A 0.000, B 0.000, C 0.000 }
gfCNCPoint6[10070] = {X 471.6054, Y 44.1516, Z -8.0000, A 0.000, B 0.000, C 0.000 }
gfCNCPoint6[10071] = {X 471.7016, Y 43.3174, Z -8.0000, A 0.000, B 0.000, C 0.000 }
gfCNCPoint6[10072] = {X 471.9634, Y 42.5195, Z -8.0000, A 0.000, B 0.000, C 0.000 }
gfCNCPoint6[10073] = {X 472.3801, Y 41.7905, Z -8.0000, A 0.000, B 0.000, C 0.000 }
gfCNCPoint6[10074] = {X 472.9347, Y 41.1600, Z -8.0000, A 0.000, B 0.000, C 0.000 }
gfCNCPoint6[10075] = {X 473.6046, Y 40.6537, Z -8.0000, A 0.000, B 0.000, C 0.000 }
gfCNCPoint6[10076] = {X 474.3626, Y 40.2923, Z -8.0000, A 0.000, B 0.000, C 0.000 }
gfCNCPoint6[10077] = {X 478.4443, Y 32.3027, Z -8.0000, A 0.000, B 0.000, C 0.000 }
gfCNCPoint6[10078] = {X 477.1665, Y 31.4492, Z -8.0000, A 0.000, B 0.000, C 0.000 }
gfCNCPoint6[10079] = {X 476.0165, Y 30.4301, Z -8.0000, A 0.000, B 0.000, C 0.000 }
gfCNCPoint6[10080] = {X 475.0154, Y 29.2643, Z -8.0000, A 0.000, B 0.000, C 0.000 }
gfCNCPoint6[10081] = {X 474.1819, Y 27.9734, Z -8.0000, A 0.000, B 0.000, C 0.000 }
gfCNCPoint6[10082] = {X 473.5313, Y 26.5813, Z -8.0000, A 0.000, B 0.000, C 0.000 }
gfCNCPoint6[10083] = {X 473.0757, Y 25.1138, Z -8.0000, A 0.000, B 0.000, C 0.000 }
gfCNCPoint6[10084] = {X 472.7651, Y 23.4467, Z -8.0000, A 0.000, B 0.000, C 0.000 }
gfCNCPoint6[10085] = {X 472.6263, Y 21.7567, Z -8.0000, A 0.000, B 0.000, C 0.000 }
gfCNCPoint6[10086] = {X 472.6607, Y 20.0613, Z -8.0000, A 0.000, B 0.000, C 0.000 }
gfCNCPoint6[10087] = {X 472.8679, Y 18.3783, Z -8.0000, A 0.000, B 0.000, C 0.000 }
gfCNCPoint6[10088] = {X 473.2458, Y 16.7252, Z -8.0000, A 0.000, B 0.000, C 0.000 }
gfCNCPoint6[10089] = {X 473.7814, Y 15.2307, Z -8.0000, A 0.000, B 0.000, C 0.000 }
gfCNCPoint6[10090] = {X 474.5149, Y 13.8227, Z -8.0000, A 0.000, B 0.000, C 0.000 }
gfCNCPoint6[10091] = {X 475.4326, Y 12.5272, Z -8.0000, A 0.000, B 0.000, C 0.000 }
gfCNCPoint6[10092] = {X 476.5176, Y 11.3682, Z -8.0000, A 0.000, B 0.000, C 0.000 }
gfCNCPoint6[10093] = {X 477.7497, Y 10.3670, Z -8.0000, A 0.000, B 0.000, C 0.000 }
gfCNCPoint6[10094] = {X 479.1063, Y 9.5423, Z -8.0000, A 0.000, B 0.000, C 0.000 }
gfCNCPoint6[10095] = {X 480.5622, Y 8.9092, Z -8.0000, A 0.000, B 0.000, C 0.000 }
gfCNCPoint6[10096] = {X 482.0905, Y 8.4795, Z -8.0000, A 0.000, B 0.000, C 0.000 }
gfCNCPoint6[10097] = {X 484.1725, Y 8.1551, Z -8.0000, A 0.000, B 0.000, C 0.000 }
gfCNCPoint6[10098] = {X 486.2765, Y 8.0414, Z -8.0000, A 0.000, B 0.000, C 0.000 }
gfCNCPoint6[10099] = {X 486.9693, Y 8.0292, Z -8.0000, A 0.000, B 0.000, C 0.000 }
gfCNCPoint6[10100] = {X 492.3835, Y 8.0292, Z -8.0000, A 0.000, B 0.000, C 0.000 }
gfCNCPoint6[10101] = {X 492.3835, Y 4.0292, Z -8.0000, A 0.000, B 0.000, C 0.000 }
gfCNCPoint6[10102] = {X 492.3835, Y 8.1092, Z -8.0000, A 0.000, B 0.000, C 0.000 }
gfCNCPoint6[10103] = {X 502.2056, Y 8.1092, Z -8.0000, A 0.000, B 0.000, C 0.000 }
gfCNCPoint6[10104] = {X 502.7375, Y 8.1134, Z -8.0000, A 0.000, B 0.000, C 0.000 }
gfCNCPoint6[10105] = {X 503.6363, Y 8.2213, Z -8.0000, A 0.000, B 0.000, C 0.000 }
gfCNCPoint6[10106] = {X 504.4889, Y 8.5255, Z -8.0000, A 0.000, B 0.000, C 0.000 }
gfCNCPoint6[10107] = {X 505.2530, Y 9.0109, Z -8.0000, A 0.000, B 0.000, C 0.000 }
gfCNCPoint6[10108] = {X 505.8906, Y 9.6535, Z -8.0000, A 0.000, B 0.000, C 0.000 }
gfCNCPoint6[10109] = {X 506.3701, Y 10.4214, Z -8.0000, A 0.000, B 0.000, C 0.000 }
gfCNCPoint6[10110] = {X 506.6676, Y 11.2763, Z -8.0000, A 0.000, B 0.000, C 0.000 }
gfCNCPoint6[10111] = {X 506.7685, Y 12.1759, Z -8.0000, A 0.000, B 0.000, C 0.000 }
gfCNCPoint6[10112] = {X 506.7685, Y 12.9782, Z -8.0000, A 0.000, B 0.000, C 0.000 }
gfCNCPoint6[10113] = {X 506.6668, Y 13.8831, Z -8.0000, A 0.000, B 0.000, C 0.000 }
gfCNCPoint6[10114] = {X 506.3670, Y 14.7429, Z -8.0000, A 0.000, B 0.000, C 0.000 }
gfCNCPoint6[10115] = {X 505.8840, Y 15.5148, Z -8.0000, A 0.000, B 0.000, C 0.000 }
gfCNCPoint6[10116] = {X 505.2418, Y 16.1603, Z -8.0000, A 0.000, B 0.000, C 0.000 }
gfCNCPoint6[10117] = {X 505.2424, Y 41.0271, Z -8.0000, A 0.000, B 0.000, C 0.000 }
gfCNCPoint6[10118] = {X 505.3173, Y 41.0885, Z -8.0000, A 0.000, B 0.000, C 0.000 }
gfCNCPoint6[10119] = {X 505.9237, Y 41.7228, Z -8.0000, A 0.000, B 0.000, C 0.000 }
gfCNCPoint6[10120] = {X 506.3804, Y 42.4721, Z -8.0000, A 0.000, B 0.000, C 0.000 }
gfCNCPoint6[10121] = {X 506.6664, Y 43.3018, Z -8.0000, A 0.000, B 0.000, C 0.000 }
gfCNCPoint6[10122] = {X 506.7683, Y 44.1734, Z -8.0000, A 0.000, B 0.000, C 0.000 }
gfCNCPoint6[10123] = {X 506.7685, Y 45.0000, Z -8.0000, A 0.000, B 0.000, C 0.000 }
gfCNCPoint6[10124] = {X 506.6662, Y 45.9079, Z -8.0000, A 0.000, B 0.000, C 0.000 }
gfCNCPoint6[10125] = {X 506.3644, Y 46.7702, Z -8.0000, A 0.000, B 0.000, C 0.000 }
gfCNCPoint6[10126] = {X 505.8784, Y 47.5438, Z -8.0000, A 0.000, B 0.000, C 0.000 }
gfCNCPoint6[10127] = {X 505.2323, Y 48.1899, Z -8.0000, A 0.000, B 0.000, C 0.000 }
gfCNCPoint6[10128] = {X 504.4587, Y 48.6760, Z -8.0000, A 0.000, B 0.000, C 0.000 }
gfCNCPoint6[10129] = {X 503.5964, Y 48.9777, Z -8.0000, A 0.000, B 0.000, C 0.000 }
gfCNCPoint6[10130] = {X 502.6885, Y 49.0800, Z -8.0000, A 0.000, B 0.000, C 0.000 }
gfCNCPoint6[10131] = {X 496.2450, Y 49.0800, Z -8.0000, A 0.000, B 0.000, C 0.000 }
gfCNCPoint6[10132] = {X 495.3416, Y 48.9787, Z -8.0000, A 0.000, B 0.000, C 0.000 }
gfCNCPoint6[10133] = {X 494.4831, Y 48.6799, Z -8.0000, A 0.000, B 0.000, C 0.000 }
gfCNCPoint6[10134] = {X 493.7120, Y 48.1985, Z -8.0000, A 0.000, B 0.000, C 0.000 }
gfCNCPoint6[10135] = {X 493.0667, Y 47.5582, Z -8.0000, A 0.000, B 0.000, C 0.000 }
gfCNCPoint6[10136] = {X 492.5791, Y 46.7909, Z -8.0000, A 0.000, B 0.000, C 0.000 }
gfCNCPoint6[10137] = {X 492.2736, Y 45.9348, Z -8.0000, A 0.000, B 0.000, C 0.000 }
gfCNCPoint6[10138] = {X 492.1652, Y 45.0322, Z -8.0000, A 0.000, B 0.000, C 0.000 }
gfCNCPoint6[10139] = {X 492.1654, Y 44.1527, Z -8.0000, A 0.000, B 0.000, C 0.000 }
gfCNCPoint6[10140] = {X 492.2760, Y 43.2637, Z -8.0000, A 0.000, B 0.000, C 0.000 }
gfCNCPoint6[10141] = {X 492.5779, Y 42.4203, Z -8.0000, A 0.000, B 0.000, C 0.000 }
gfCNCPoint6[10142] = {X 493.0566, Y 41.6631, Z -8.0000, A 0.000, B 0.000, C 0.000 }
gfCNCPoint6[10143] = {X 493.6890, Y 41.0287, Z -8.0000, A 0.000, B 0.000, C 0.000 }
gfCNCPoint6[10144] = {X 493.6890, Y 34.2338, Z -8.0000, A 0.000, B 0.000, C 0.000 }
gfCNCPoint6[10145] = {X 490.5792, Y 34.2338, Z -8.0000, A 0.000, B 0.000, C 0.000 }
gfCNCPoint6[10146] = {X 486.1793, Y 42.8021, Z -8.0000, A 0.000, B 0.000, C 0.000 }
gfCNCPoint6[10147] = {X 486.2190, Y 42.9106, Z -8.0000, A 0.000, B 0.000, C 0.000 }
gfCNCPoint6[10148] = {X 486.3747, Y 43.5330, Z -8.0000, A 0.000, B 0.000, C 0.000 }
gfCNCPoint6[10149] = {X 486.4309, Y 44.1720, Z -8.0000, A 0.000, B 0.000, C 0.000 }
gfCNCPoint6[10150] = {X 486.4310, Y 45.0000, Z -8.0000, A 0.000, B 0.000, C 0.000 }
gfCNCPoint6[10151] = {X 486.3287, Y 45.9079, Z -8.0000, A 0.000, B 0.000, C 0.000 }
gfCNCPoint6[10152] = {X 486.0270, Y 46.7702, Z -8.0000, A 0.000, B 0.000, C 0.000 }
gfCNCPoint6[10153] = {X 485.5409, Y 47.5438, Z -8.0000, A 0.000, B 0.000, C 0.000 }
gfCNCPoint6[10154] = {X 484.8949, Y 48.1899, Z -8.0000, A 0.000, B 0.000, C 0.000 }
gfCNCPoint6[10155] = {X 484.1213, Y 48.6760, Z -8.0000, A 0.000, B 0.000, C 0.000 }
gfCNCPoint6[10156] = {X 483.2589, Y 48.9777, Z -8.0000, A 0.000, B 0.000, C 0.000 }
gfCNCPoint6[10157] = {X 482.3510, Y 49.0800, Z -8.0000, A 0.000, B 0.000, C 0.000 }
gfCNCPoint6[10158] = {X 475.7650, Y 49.0800, Z -8.0000, A 0.000, B 0.000, C 0.000 }
gfCNCPoint6[10159] = {X 474.8571, Y 48.9777, Z -8.0000, A 0.000, B 0.000, C 0.000 }
gfCNCPoint6[10160] = {X 473.9947, Y 48.6760, Z -8.0000, A 0.000, B 0.000, C 0.000 }
gfCNCPoint6[10161] = {X 473.2211, Y 48.1899, Z -8.0000, A 0.000, B 0.000, C 0.000 }
gfCNCPoint6[10162] = {X 472.5751, Y 47.5438, Z -8.0000, A 0.000, B 0.000, C 0.000 }
gfCNCPoint6[10163] = {X 472.0890, Y 46.7702, Z -8.0000, A 0.000, B 0.000, C 0.000 }
gfCNCPoint6[10164] = {X 471.7873, Y 45.9079, Z -8.0000, A 0.000, B 0.000, C 0.000 }
gfCNCPoint6[10165] = {X 471.6850, Y 45.0000, Z -8.0000, A 0.000, B 0.000, C 0.000 }
gfCNCPoint6[10166] = {X 471.6853, Y 44.1527, Z -8.0000, A 0.000, B 0.000, C 0.000 }
gfCNCPoint6[10167] = {X 471.7809, Y 43.3294, Z -8.0000, A 0.000, B 0.000, C 0.000 }
gfCNCPoint6[10168] = {X 472.0408, Y 42.5424, Z -8.0000, A 0.000, B 0.000, C 0.000 }
gfCNCPoint6[10169] = {X 472.4544, Y 41.8242, Z -8.0000, A 0.000, B 0.000, C 0.000 }
gfCNCPoint6[10170] = {X 473.0046, Y 41.2044, Z -8.0000, A 0.000, B 0.000, C 0.000 }
gfCNCPoint6[10171] = {X 473.6687, Y 40.7085, Z -8.0000, A 0.000, B 0.000, C 0.000 }
gfCNCPoint6[10172] = {X 474.4193, Y 40.3571, Z -8.0000, A 0.000, B 0.000, C 0.000 }
gfCNCPoint6[10173] = {X 478.5503, Y 32.2710, Z -8.0000, A 0.000, B 0.000, C 0.000 }
gfCNCPoint6[10174] = {X 477.2658, Y 31.4245, Z -8.0000, A 0.000, B 0.000, C 0.000 }
gfCNCPoint6[10175] = {X 476.1092, Y 30.4100, Z -8.0000, A 0.000, B 0.000, C 0.000 }
gfCNCPoint6[10176] = {X 475.1023, Y 29.2469, Z -8.0000, A 0.000, B 0.000, C 0.000 }
gfCNCPoint6[10177] = {X 474.2641, Y 27.9568, Z -8.0000, A 0.000, B 0.000, C 0.000 }
gfCNCPoint6[10178] = {X 473.6104, Y 26.5642, Z -8.0000, A 0.000, B 0.000, C 0.000 }
gfCNCPoint6[10179] = {X 473.1535, Y 25.0952, Z -8.0000, A 0.000, B 0.000, C 0.000 }
gfCNCPoint6[10180] = {X 472.8444, Y 23.4361, Z -8.0000, A 0.000, B 0.000, C 0.000 }
gfCNCPoint6[10181] = {X 472.7063, Y 21.7542, Z -8.0000, A 0.000, B 0.000, C 0.000 }
gfCNCPoint6[10182] = {X 472.7405, Y 20.0670, Z -8.0000, A 0.000, B 0.000, C 0.000 }
gfCNCPoint6[10183] = {X 472.9467, Y 18.3921, Z -8.0000, A 0.000, B 0.000, C 0.000 }
gfCNCPoint6[10184] = {X 473.3227, Y 16.7470, Z -8.0000, A 0.000, B 0.000, C 0.000 }
gfCNCPoint6[10185] = {X 473.8548, Y 15.2627, Z -8.0000, A 0.000, B 0.000, C 0.000 }
gfCNCPoint6[10186] = {X 474.5832, Y 13.8644, Z -8.0000, A 0.000, B 0.000, C 0.000 }
gfCNCPoint6[10187] = {X 475.4946, Y 12.5777, Z -8.0000, A 0.000, B 0.000, C 0.000 }
gfCNCPoint6[10188] = {X 476.5721, Y 11.4267, Z -8.0000, A 0.000, B 0.000, C 0.000 }
gfCNCPoint6[10189] = {X 477.7958, Y 10.4324, Z -8.0000, A 0.000, B 0.000, C 0.000 }
gfCNCPoint6[10190] = {X 479.1431, Y 9.6133, Z -8.0000, A 0.000, B 0.000, C 0.000 }
gfCNCPoint6[10191] = {X 480.5891, Y 8.9846, Z -8.0000, A 0.000, B 0.000, C 0.000 }
gfCNCPoint6[10192] = {X 482.1069, Y 8.5578, Z -8.0000, A 0.000, B 0.000, C 0.000 }
gfCNCPoint6[10193] = {X 484.1811, Y 8.2347, Z -8.0000, A 0.000, B 0.000, C 0.000 }
gfCNCPoint6[10194] = {X 486.2773, Y 8.1214, Z -8.0000, A 0.000, B 0.000, C 0.000 }
gfCNCPoint6[10195] = {X 486.9700, Y 8.1092, Z -8.0000, A 0.000, B 0.000, C 0.000 }
gfCNCPoint6[10196] = {X 492.3835, Y 8.1092, Z -8.0000, A 0.000, B 0.000, C 0.000 }
gfCNCPoint6[10197] = {X 492.3835, Y 4.1092, Z -8.0000, A 0.000, B 0.000, C 0.000 }
gfCNCPoint6[10198] = {X 492.3835, Y 8.1892, Z -8.0000, A 0.000, B 0.000, C 0.000 }
gfCNCPoint6[10199] = {X 502.2053, Y 8.1892, Z -8.0000, A 0.000, B 0.000, C 0.000 }
gfCNCPoint6[10200] = {X 502.7369, Y 8.1934, Z -8.0000, A 0.000, B 0.000, C 0.000 }
gfCNCPoint6[10201] = {X 503.6180, Y 8.2991, Z -8.0000, A 0.000, B 0.000, C 0.000 }
gfCNCPoint6[10202] = {X 504.4538, Y 8.5974, Z -8.0000, A 0.000, B 0.000, C 0.000 }
gfCNCPoint6[10203] = {X 505.2028, Y 9.0733, Z -8.0000, A 0.000, B 0.000, C 0.000 }
gfCNCPoint6[10204] = {X 505.8279, Y 9.7032, Z -8.0000, A 0.000, B 0.000, C 0.000 }
gfCNCPoint6[10205] = {X 506.2979, Y 10.4559, Z -8.0000, A 0.000, B 0.000, C 0.000 }
gfCNCPoint6[10206] = {X 506.5896, Y 11.2940, Z -8.0000, A 0.000, B 0.000, C 0.000 }
gfCNCPoint6[10207] = {X 506.6885, Y 12.1759, Z -8.0000, A 0.000, B 0.000, C 0.000 }
gfCNCPoint6[10208] = {X 506.6883, Y 13.0192, Z -8.0000, A 0.000, B 0.000, C 0.000 }
gfCNCPoint6[10209] = {X 506.5797, Y 13.9046, Z -8.0000, A 0.000, B 0.000, C 0.000 }
gfCNCPoint6[10210] = {X 506.2776, Y 14.7439, Z -8.0000, A 0.000, B 0.000, C 0.000 }
gfCNCPoint6[10211] = {X 505.7970, Y 15.4954, Z -8.0000, A 0.000, B 0.000, C 0.000 }
gfCNCPoint6[10212] = {X 505.1618, Y 16.1217, Z -8.0000, A 0.000, B 0.000, C 0.000 }
gfCNCPoint6[10213] = {X 505.1624, Y 41.0649, Z -8.0000, A 0.000, B 0.000, C 0.000 }
gfCNCPoint6[10214] = {X 505.3011, Y 41.1799, Z -8.0000, A 0.000, B 0.000, C 0.000 }
gfCNCPoint6[10215] = {X 505.8866, Y 41.8063, Z -8.0000, A 0.000, B 0.000, C 0.000 }
gfCNCPoint6[10216] = {X 506.3252, Y 42.5431, Z -8.0000, A 0.000, B 0.000, C 0.000 }
gfCNCPoint6[10217] = {X 506.5966, Y 43.3564, Z -8.0000, A 0.000, B 0.000, C 0.000 }
gfCNCPoint6[10218] = {X 506.6885, Y 44.2089, Z -8.0000, A 0.000, B 0.000, C 0.000 }
gfCNCPoint6[10219] = {X 506.6885, Y 45.0000, Z -8.0000, A 0.000, B 0.000, C 0.000 }
gfCNCPoint6[10220] = {X 506.5882, Y 45.8901, Z -8.0000, A 0.000, B 0.000, C 0.000 }
gfCNCPoint6[10221] = {X 506.2924, Y 46.7355, Z -8.0000, A 0.000, B 0.000, C 0.000 }
gfCNCPoint6[10222] = {X 505.8158, Y 47.4940, Z -8.0000, A 0.000, B 0.000, C 0.000 }
gfCNCPoint6[10223] = {X 505.1825, Y 48.1273, Z -8.0000, A 0.000, B 0.000, C 0.000 }
gfCNCPoint6[10224] = {X 504.4240, Y 48.6039, Z -8.0000, A 0.000, B 0.000, C 0.000 }
gfCNCPoint6[10225] = {X 503.5786, Y 48.8997, Z -8.0000, A 0.000, B 0.000, C 0.000 }
gfCNCPoint6[10226] = {X 502.6885, Y 49.0000, Z -8.0000, A 0.000, B 0.000, C 0.000 }
gfCNCPoint6[10227] = {X 496.2450, Y 49.0000, Z -8.0000, A 0.000, B 0.000, C 0.000 }
gfCNCPoint6[10228] = {X 495.3549, Y 48.8997, Z -8.0000, A 0.000, B 0.000, C 0.000 }
gfCNCPoint6[10229] = {X 494.5095, Y 48.6039, Z -8.0000, A 0.000, B 0.000, C 0.000 }
gfCNCPoint6[10230] = {X 493.7511, Y 48.1273, Z -8.0000, A 0.000, B 0.000, C 0.000 }
gfCNCPoint6[10231] = {X 493.1177, Y 47.4939, Z -8.0000, A 0.000, B 0.000, C 0.000 }
gfCNCPoint6[10232] = {X 492.6411, Y 46.7355, Z -8.0000, A 0.000, B 0.000, C 0.000 }
gfCNCPoint6[10233] = {X 492.3453, Y 45.8901, Z -8.0000, A 0.000, B 0.000, C 0.000 }
gfCNCPoint6[10234] = {X 492.2450, Y 45.0000, Z -8.0000, A 0.000, B 0.000, C 0.000 }
gfCNCPoint6[10235] = {X 492.2454, Y 44.1538, Z -8.0000, A 0.000, B 0.000, C 0.000 }
gfCNCPoint6[10236] = {X 492.3560, Y 43.2730, Z -8.0000, A 0.000, B 0.000, C 0.000 }
gfCNCPoint6[10237] = {X 492.6582, Y 42.4382, Z -8.0000, A 0.000, B 0.000, C 0.000 }
gfCNCPoint6[10238] = {X 493.1371, Y 41.6907, Z -8.0000, A 0.000, B 0.000, C 0.000 }
gfCNCPoint6[10239] = {X 493.7690, Y 41.0672, Z -8.0000, A 0.000, B 0.000, C 0.000 }
gfCNCPoint6[10240] = {X 493.7690, Y 34.1538, Z -8.0000, A 0.000, B 0.000, C 0.000 }
gfCNCPoint6[10241] = {X 490.7746, Y 34.1538, Z -8.0000, A 0.000, B 0.000, C 0.000 }
gfCNCPoint6[10242] = {X 490.5309, Y 34.1527, Z -8.0000, A 0.000, B 0.000, C 0.000 }
gfCNCPoint6[10243] = {X 486.0921, Y 42.7967, Z -8.0000, A 0.000, B 0.000, C 0.000 }
gfCNCPoint6[10244] = {X 486.1479, Y 42.9503, Z -8.0000, A 0.000, B 0.000, C 0.000 }
gfCNCPoint6[10245] = {X 486.2999, Y 43.5714, Z -8.0000, A 0.000, B 0.000, C 0.000 }
gfCNCPoint6[10246] = {X 486.3510, Y 44.2089, Z -8.0000, A 0.000, B 0.000, C 0.000 }
gfCNCPoint6[10247] = {X 486.3510, Y 45.0000, Z -8.0000, A 0.000, B 0.000, C 0.000 }
gfCNCPoint6[10248] = {X 486.2507, Y 45.8901, Z -8.0000, A 0.000, B 0.000, C 0.000 }
gfCNCPoint6[10249] = {X 485.9549, Y 46.7355, Z -8.0000, A 0.000, B 0.000, C 0.000 }
gfCNCPoint6[10250] = {X 485.4783, Y 47.4940, Z -8.0000, A 0.000, B 0.000, C 0.000 }
gfCNCPoint6[10251] = {X 484.8450, Y 48.1273, Z -8.0000, A 0.000, B 0.000, C 0.000 }
gfCNCPoint6[10252] = {X 484.0866, Y 48.6039, Z -8.0000, A 0.000, B 0.000, C 0.000 }
gfCNCPoint6[10253] = {X 483.2411, Y 48.8997, Z -8.0000, A 0.000, B 0.000, C 0.000 }
gfCNCPoint6[10254] = {X 482.3510, Y 49.0000, Z -8.0000, A 0.000, B 0.000, C 0.000 }
gfCNCPoint6[10255] = {X 475.7650, Y 49.0000, Z -8.0000, A 0.000, B 0.000, C 0.000 }
gfCNCPoint6[10256] = {X 474.8749, Y 48.8997, Z -8.0000, A 0.000, B 0.000, C 0.000 }
gfCNCPoint6[10257] = {X 474.0294, Y 48.6039, Z -8.0000, A 0.000, B 0.000, C 0.000 }
gfCNCPoint6[10258] = {X 473.2710, Y 48.1273, Z -8.0000, A 0.000, B 0.000, C 0.000 }
gfCNCPoint6[10259] = {X 472.6376, Y 47.4940, Z -8.0000, A 0.000, B 0.000, C 0.000 }
gfCNCPoint6[10260] = {X 472.1611, Y 46.7355, Z -8.0000, A 0.000, B 0.000, C 0.000 }
gfCNCPoint6[10261] = {X 471.8652, Y 45.8901, Z -8.0000, A 0.000, B 0.000, C 0.000 }
gfCNCPoint6[10262] = {X 471.7650, Y 45.0000, Z -8.0000, A 0.000, B 0.000, C 0.000 }
gfCNCPoint6[10263] = {X 471.7653, Y 44.1538, Z -8.0000, A 0.000, B 0.000, C 0.000 }
gfCNCPoint6[10264] = {X 471.8601, Y 43.3414, Z -8.0000, A 0.000, B 0.000, C 0.000 }
gfCNCPoint6[10265] = {X 472.1182, Y 42.5654, Z -8.0000, A 0.000, B 0.000, C 0.000 }
gfCNCPoint6[10266] = {X 472.5286, Y 41.8580, Z -8.0000, A 0.000, B 0.000, C 0.000 }
gfCNCPoint6[10267] = {X 473.0744, Y 41.2489, Z -8.0000, A 0.000, B 0.000, C 0.000 }
gfCNCPoint6[10268] = {X 473.7327, Y 40.7635, Z -8.0000, A 0.000, B 0.000, C 0.000 }
gfCNCPoint6[10269] = {X 474.4759, Y 40.4222, Z -8.0000, A 0.000, B 0.000, C 0.000 }
gfCNCPoint6[10270] = {X 478.6566, Y 32.2388, Z -8.0000, A 0.000, B 0.000, C 0.000 }
gfCNCPoint6[10271] = {X 477.3652, Y 31.3994, Z -8.0000, A 0.000, B 0.000, C 0.000 }
gfCNCPoint6[10272] = {X 476.2020, Y 30.3898, Z -8.0000, A 0.000, B 0.000, C 0.000 }
gfCNCPoint6[10273] = {X 475.1893, Y 29.2293, Z -8.0000, A 0.000, B 0.000, C 0.000 }
gfCNCPoint6[10274] = {X 474.3465, Y 27.9402, Z -8.0000, A 0.000, B 0.000, C 0.000 }
gfCNCPoint6[10275] = {X 473.6896, Y 26.5470, Z -8.0000, A 0.000, B 0.000, C 0.000 }
gfCNCPoint6[10276] = {X 473.2313, Y 25.0766, Z -8.0000, A 0.000, B 0.000, C 0.000 }
gfCNCPoint6[10277] = {X 472.9237, Y 23.4256, Z -8.0000, A 0.000, B 0.000, C 0.000 }
gfCNCPoint6[10278] = {X 472.7862, Y 21.7518, Z -8.0000, A 0.000, B 0.000, C 0.000 }
gfCNCPoint6[10279] = {X 472.8203, Y 20.0727, Z -8.0000, A 0.000, B 0.000, C 0.000 }
gfCNCPoint6[10280] = {X 473.0255, Y 18.4059, Z -8.0000, A 0.000, B 0.000, C 0.000 }
gfCNCPoint6[10281] = {X 473.3997, Y 16.7687, Z -8.0000, A 0.000, B 0.000, C 0.000 }
gfCNCPoint6[10282] = {X 473.9281, Y 15.2947, Z -8.0000, A 0.000, B 0.000, C 0.000 }
gfCNCPoint6[10283] = {X 474.6515, Y 13.9060, Z -8.0000, A 0.000, B 0.000, C 0.000 }
gfCNCPoint6[10284] = {X 475.5566, Y 12.6283, Z -8.0000, A 0.000, B 0.000, C 0.000 }
gfCNCPoint6[10285] = {X 476.6267, Y 11.4852, Z -8.0000, A 0.000, B 0.000, C 0.000 }
gfCNCPoint6[10286] = {X 477.8420, Y 10.4978, Z -8.0000, A 0.000, B 0.000, C 0.000 }
gfCNCPoint6[10287] = {X 479.1799, Y 9.6844, Z -8.0000, A 0.000, B 0.000, C 0.000 }
gfCNCPoint6[10288] = {X 480.6159, Y 9.0600, Z -8.0000, A 0.000, B 0.000, C 0.000 }
gfCNCPoint6[10289] = {X 482.1233, Y 8.6361, Z -8.0000, A 0.000, B 0.000, C 0.000 }
gfCNCPoint6[10290] = {X 484.1898, Y 8.3142, Z -8.0000, A 0.000, B 0.000, C 0.000 }
gfCNCPoint6[10291] = {X 486.2782, Y 8.2014, Z -8.0000, A 0.000, B 0.000, C 0.000 }
gfCNCPoint6[10292] = {X 486.9707, Y 8.1892, Z -8.0000, A 0.000, B 0.000, C 0.000 }
gfCNCPoint6[10293] = {X 492.3835, Y 8.1892, Z -8.0000, A 0.000, B 0.000, C 0.000 }
gfCNCPoint6[10294] = {X 492.3835, Y 4.1092, Z -8.0000, A 0.000, B 0.000, C 0.000 }
gfCNCPoint6[10295] = {X 492.3835, Y 4.1092, Z -5.0000, A 0.000, B 0.000, C 0.000 }
gfCNCPoint6[10296] = {X 492.3835, Y 4.1092, Z 11.0000, A 0.000, B 0.000, C 0.000 }
gfCNCPoint6[10297] = {X 533.9633, Y 3.7892, Z 11.0000, A 0.000, B 0.000, C 0.000 }
gfCNCPoint6[10298] = {X 533.9633, Y 3.7892, Z -5.0000, A 0.000, B 0.000, C 0.000 }
gfCNCPoint6[10299] = {X 533.9633, Y 3.7892, Z -8.0000, A 0.000, B 0.000, C 0.000 }
gfCNCPoint6[10300] = {X 533.9633, Y 7.8692, Z -8.0000, A 0.000, B 0.000, C 0.000 }
gfCNCPoint6[10301] = {X 543.7499, Y 7.8692, Z -8.0000, A 0.000, B 0.000, C 0.000 }
gfCNCPoint6[10302] = {X 544.7304, Y 7.9548, Z -8.0000, A 0.000, B 0.000, C 0.000 }
gfCNCPoint6[10303] = {X 545.6661, Y 8.2597, Z -8.0000, A 0.000, B 0.000, C 0.000 }
gfCNCPoint6[10304] = {X 546.5086, Y 8.7684, Z -8.0000, A 0.000, B 0.000, C 0.000 }
gfCNCPoint6[10305] = {X 547.2143, Y 9.4543, Z -8.0000, A 0.000, B 0.000, C 0.000 }
gfCNCPoint6[10306] = {X 547.7467, Y 10.2821, Z -8.0000, A 0.000, B 0.000, C 0.000 }
gfCNCPoint6[10307] = {X 548.0781, Y 11.2088, Z -8.0000, A 0.000, B 0.000, C 0.000 }
gfCNCPoint6[10308] = {X 548.1914, Y 12.1864, Z -8.0000, A 0.000, B 0.000, C 0.000 }
gfCNCPoint6[10309] = {X 548.1912, Y 13.0225, Z -8.0000, A 0.000, B 0.000, C 0.000 }
gfCNCPoint6[10310] = {X 548.0830, Y 13.9400, Z -8.0000, A 0.000, B 0.000, C 0.000 }
gfCNCPoint6[10311] = {X 547.7821, Y 14.8135, Z -8.0000, A 0.000, B 0.000, C 0.000 }
gfCNCPoint6[10312] = {X 547.3024, Y 15.6031, Z -8.0000, A 0.000, B 0.000, C 0.000 }
gfCNCPoint6[10313] = {X 546.6658, Y 16.2726, Z -8.0000, A 0.000, B 0.000, C 0.000 }
gfCNCPoint6[10314] = {X 546.6653, Y 40.9144, Z -8.0000, A 0.000, B 0.000, C 0.000 }
gfCNCPoint6[10315] = {X 546.6870, Y 40.9323, Z -8.0000, A 0.000, B 0.000, C 0.000 }
gfCNCPoint6[10316] = {X 547.3164, Y 41.6022, Z -8.0000, A 0.000, B 0.000, C 0.000 }
gfCNCPoint6[10317] = {X 547.7899, Y 42.3900, Z -8.0000, A 0.000, B 0.000, C 0.000 }
gfCNCPoint6[10318] = {X 548.0860, Y 43.2602, Z -8.0000, A 0.000, B 0.000, C 0.000 }
gfCNCPoint6[10319] = {X 548.1913, Y 44.1733, Z -8.0000, A 0.000, B 0.000, C 0.000 }
gfCNCPoint6[10320] = {X 548.1914, Y 45.0004, Z -8.0000, A 0.000, B 0.000, C 0.000 }
gfCNCPoint6[10321] = {X 548.0781, Y 45.9780, Z -8.0000, A 0.000, B 0.000, C 0.000 }
gfCNCPoint6[10322] = {X 547.7466, Y 46.9047, Z -8.0000, A 0.000, B 0.000, C 0.000 }
gfCNCPoint6[10323] = {X 547.2143, Y 47.7324, Z -8.0000, A 0.000, B 0.000, C 0.000 }
gfCNCPoint6[10324] = {X 546.5085, Y 48.4183, Z -8.0000, A 0.000, B 0.000, C 0.000 }
gfCNCPoint6[10325] = {X 545.6660, Y 48.9269, Z -8.0000, A 0.000, B 0.000, C 0.000 }
gfCNCPoint6[10326] = {X 544.7303, Y 49.2318, Z -8.0000, A 0.000, B 0.000, C 0.000 }
gfCNCPoint6[10327] = {X 543.7499, Y 49.3173, Z -8.0000, A 0.000, B 0.000, C 0.000 }
gfCNCPoint6[10328] = {X 524.0457, Y 49.3176, Z -8.0000, A 0.000, B 0.000, C 0.000 }
gfCNCPoint6[10329] = {X 523.4990, Y 49.9514, Z -8.0000, A 0.000, B 0.000, C 0.000 }
gfCNCPoint6[10330] = {X 522.8439, Y 50.4724, Z -8.0000, A 0.000, B 0.000, C 0.000 }
gfCNCPoint6[10331] = {X 522.1032, Y 50.8622, Z -8.0000, A 0.000, B 0.000, C 0.000 }
gfCNCPoint6[10332] = {X 521.3028, Y 51.1073, Z -8.0000, A 0.000, B 0.000, C 0.000 }
gfCNCPoint6[10333] = {X 520.4708, Y 51.1991, Z -8.0000, A 0.000, B 0.000, C 0.000 }
gfCNCPoint6[10334] = {X 519.7998, Y 51.1991, Z -8.0000, A 0.000, B 0.000, C 0.000 }
gfCNCPoint6[10335] = {X 518.8385, Y 51.0908, Z -8.0000, A 0.000, B 0.000, C 0.000 }
gfCNCPoint6[10336] = {X 517.9254, Y 50.7713, Z -8.0000, A 0.000, B 0.000, C 0.000 }
gfCNCPoint6[10337] = {X 517.1063, Y 50.2566, Z -8.0000, A 0.000, B 0.000, C 0.000 }
gfCNCPoint6[10338] = {X 516.4223, Y 49.5726, Z -8.0000, A 0.000, B 0.000, C 0.000 }
gfCNCPoint6[10339] = {X 515.9076, Y 48.7535, Z -8.0000, A 0.000, B 0.000, C 0.000 }
gfCNCPoint6[10340] = {X 515.5881, Y 47.8404, Z -8.0000, A 0.000, B 0.000, C 0.000 }
gfCNCPoint6[10341] = {X 515.4798, Y 46.8791, Z -8.0000, A 0.000, B 0.000, C 0.000 }
gfCNCPoint6[10342] = {X 515.4798, Y 39.9011, Z -8.0000, A 0.000, B 0.000, C 0.000 }
gfCNCPoint6[10343] = {X 515.5869, Y 38.9451, Z -8.0000, A 0.000, B 0.000, C 0.000 }
gfCNCPoint6[10344] = {X 515.9029, Y 38.0365, Z -8.0000, A 0.000, B 0.000, C 0.000 }
gfCNCPoint6[10345] = {X 516.4121, Y 37.2204, Z -8.0000, A 0.000, B 0.000, C 0.000 }
gfCNCPoint6[10346] = {X 517.0893, Y 36.5372, Z -8.0000, A 0.000, B 0.000, C 0.000 }
gfCNCPoint6[10347] = {X 517.9010, Y 36.0208, Z -8.0000, A 0.000, B 0.000, C 0.000 }
gfCNCPoint6[10348] = {X 518.8067, Y 35.6968, Z -8.0000, A 0.000, B 0.000, C 0.000 }
gfCNCPoint6[10349] = {X 519.7617, Y 35.5813, Z -8.0000, A 0.000, B 0.000, C 0.000 }
gfCNCPoint6[10350] = {X 520.5269, Y 35.5815, Z -8.0000, A 0.000, B 0.000, C 0.000 }
gfCNCPoint6[10351] = {X 521.3531, Y 35.6727, Z -8.0000, A 0.000, B 0.000, C 0.000 }
gfCNCPoint6[10352] = {X 522.1466, Y 35.9205, Z -8.0000, A 0.000, B 0.000, C 0.000 }
gfCNCPoint6[10353] = {X 522.8780, Y 36.3157, Z -8.0000, A 0.000, B 0.000, C 0.000 }
gfCNCPoint6[10354] = {X 523.5201, Y 36.8436, Z -8.0000, A 0.000, B 0.000, C 0.000 }
gfCNCPoint6[10355] = {X 524.0492, Y 37.4848, Z -8.0000, A 0.000, B 0.000, C 0.000 }
gfCNCPoint6[10356] = {X 534.6319, Y 37.4848, Z -8.0000, A 0.000, B 0.000, C 0.000 }
gfCNCPoint6[10357] = {X 534.6319, Y 33.9664, Z -8.0000, A 0.000, B 0.000, C 0.000 }
gfCNCPoint6[10358] = {X 530.1082, Y 33.9677, Z -8.0000, A 0.000, B 0.000, C 0.000 }
gfCNCPoint6[10359] = {X 529.5760, Y 34.6113, Z -8.0000, A 0.000, B 0.000, C 0.000 }
gfCNCPoint6[10360] = {X 528.9299, Y 35.1405, Z -8.0000, A 0.000, B 0.000, C 0.000 }
gfCNCPoint6[10361] = {X 528.1940, Y 35.5354, Z -8.0000, A 0.000, B 0.000, C 0.000 }
gfCNCPoint6[10362] = {X 527.3960, Y 35.7814, Z -8.0000, A 0.000, B 0.000, C 0.000 }
gfCNCPoint6[10363] = {X 526.5655, Y 35.8693, Z -8.0000, A 0.000, B 0.000, C 0.000 }
gfCNCPoint6[10364] = {X 525.8868, Y 35.8694, Z -8.0000, A 0.000, B 0.000, C 0.000 }
gfCNCPoint6[10365] = {X 524.9255, Y 35.7611, Z -8.0000, A 0.000, B 0.000, C 0.000 }
gfCNCPoint6[10366] = {X 524.0124, Y 35.4416, Z -8.0000, A 0.000, B 0.000, C 0.000 }
gfCNCPoint6[10367] = {X 523.1933, Y 34.9270, Z -8.0000, A 0.000, B 0.000, C 0.000 }
gfCNCPoint6[10368] = {X 522.5092, Y 34.2429, Z -8.0000, A 0.000, B 0.000, C 0.000 }
gfCNCPoint6[10369] = {X 521.9946, Y 33.4238, Z -8.0000, A 0.000, B 0.000, C 0.000 }
gfCNCPoint6[10370] = {X 521.6751, Y 32.5107, Z -8.0000, A 0.000, B 0.000, C 0.000 }
gfCNCPoint6[10371] = {X 521.5668, Y 31.5495, Z -8.0000, A 0.000, B 0.000, C 0.000 }
gfCNCPoint6[10372] = {X 521.5668, Y 24.5714, Z -8.0000, A 0.000, B 0.000, C 0.000 }
gfCNCPoint6[10373] = {X 521.6739, Y 23.6153, Z -8.0000, A 0.000, B 0.000, C 0.000 }
gfCNCPoint6[10374] = {X 521.9900, Y 22.7066, Z -8.0000, A 0.000, B 0.000, C 0.000 }
gfCNCPoint6[10375] = {X 522.4994, Y 21.8904, Z -8.0000, A 0.000, B 0.000, C 0.000 }
gfCNCPoint6[10376] = {X 523.1768, Y 21.2071, Z -8.0000, A 0.000, B 0.000, C 0.000 }
gfCNCPoint6[10377] = {X 523.9886, Y 20.6908, Z -8.0000, A 0.000, B 0.000, C 0.000 }
gfCNCPoint6[10378] = {X 524.8946, Y 20.3669, Z -8.0000, A 0.000, B 0.000, C 0.000 }
gfCNCPoint6[10379] = {X 525.8498, Y 20.2516, Z -8.0000, A 0.000, B 0.000, C 0.000 }
gfCNCPoint6[10380] = {X 526.5695, Y 20.2516, Z -8.0000, A 0.000, B 0.000, C 0.000 }
gfCNCPoint6[10381] = {X 527.3943, Y 20.3391, Z -8.0000, A 0.000, B 0.000, C 0.000 }
gfCNCPoint6[10382] = {X 528.1871, Y 20.5826, Z -8.0000, A 0.000, B 0.000, C 0.000 }
gfCNCPoint6[10383] = {X 528.9189, Y 20.9731, Z -8.0000, A 0.000, B 0.000, C 0.000 }
gfCNCPoint6[10384] = {X 529.5625, Y 21.4962, Z -8.0000, A 0.000, B 0.000, C 0.000 }
gfCNCPoint6[10385] = {X 530.0943, Y 22.1327, Z -8.0000, A 0.000, B 0.000, C 0.000 }
gfCNCPoint6[10386] = {X 534.6319, Y 22.1327, Z -8.0000, A 0.000, B 0.000, C 0.000 }
gfCNCPoint6[10387] = {X 534.6319, Y 19.7028, Z -8.0000, A 0.000, B 0.000, C 0.000 }
gfCNCPoint6[10388] = {X 524.1913, Y 19.7028, Z -8.0000, A 0.000, B 0.000, C 0.000 }
gfCNCPoint6[10389] = {X 523.6589, Y 20.3470, Z -8.0000, A 0.000, B 0.000, C 0.000 }
gfCNCPoint6[10390] = {X 523.0123, Y 20.8767, Z -8.0000, A 0.000, B 0.000, C 0.000 }
gfCNCPoint6[10391] = {X 522.2759, Y 21.2719, Z -8.0000, A 0.000, B 0.000, C 0.000 }
gfCNCPoint6[10392] = {X 521.4772, Y 21.5179, Z -8.0000, A 0.000, B 0.000, C 0.000 }
gfCNCPoint6[10393] = {X 520.6460, Y 21.6056, Z -8.0000, A 0.000, B 0.000, C 0.000 }
gfCNCPoint6[10394] = {X 519.9691, Y 21.6057, Z -8.0000, A 0.000, B 0.000, C 0.000 }
gfCNCPoint6[10395] = {X 519.0078, Y 21.4974, Z -8.0000, A 0.000, B 0.000, C 0.000 }
gfCNCPoint6[10396] = {X 518.0947, Y 21.1779, Z -8.0000, A 0.000, B 0.000, C 0.000 }
gfCNCPoint6[10397] = {X 517.2756, Y 20.6632, Z -8.0000, A 0.000, B 0.000, C 0.000 }
gfCNCPoint6[10398] = {X 516.5916, Y 19.9792, Z -8.0000, A 0.000, B 0.000, C 0.000 }
gfCNCPoint6[10399] = {X 516.0769, Y 19.1601, Z -8.0000, A 0.000, B 0.000, C 0.000 }
gfCNCPoint6[10400] = {X 515.7574, Y 18.2470, Z -8.0000, A 0.000, B 0.000, C 0.000 }
gfCNCPoint6[10401] = {X 515.6491, Y 17.2857, Z -8.0000, A 0.000, B 0.000, C 0.000 }
gfCNCPoint6[10402] = {X 515.6491, Y 10.3077, Z -8.0000, A 0.000, B 0.000, C 0.000 }
gfCNCPoint6[10403] = {X 515.7562, Y 9.3519, Z -8.0000, A 0.000, B 0.000, C 0.000 }
gfCNCPoint6[10404] = {X 516.0720, Y 8.4435, Z -8.0000, A 0.000, B 0.000, C 0.000 }
gfCNCPoint6[10405] = {X 516.5811, Y 7.6275, Z -8.0000, A 0.000, B 0.000, C 0.000 }
gfCNCPoint6[10406] = {X 517.2580, Y 6.9443, Z -8.0000, A 0.000, B 0.000, C 0.000 }
gfCNCPoint6[10407] = {X 518.0693, Y 6.4278, Z -8.0000, A 0.000, B 0.000, C 0.000 }
gfCNCPoint6[10408] = {X 518.9748, Y 6.1037, Z -8.0000, A 0.000, B 0.000, C 0.000 }
gfCNCPoint6[10409] = {X 519.9296, Y 5.9879, Z -8.0000, A 0.000, B 0.000, C 0.000 }
gfCNCPoint6[10410] = {X 520.6502, Y 5.9879, Z -8.0000, A 0.000, B 0.000, C 0.000 }
gfCNCPoint6[10411] = {X 521.4754, Y 6.0751, Z -8.0000, A 0.000, B 0.000, C 0.000 }
gfCNCPoint6[10412] = {X 522.2687, Y 6.3185, Z -8.0000, A 0.000, B 0.000, C 0.000 }
gfCNCPoint6[10413] = {X 523.0008, Y 6.7091, Z -8.0000, A 0.000, B 0.000, C 0.000 }
gfCNCPoint6[10414] = {X 523.6448, Y 7.2324, Z -8.0000, A 0.000, B 0.000, C 0.000 }
gfCNCPoint6[10415] = {X 524.1768, Y 7.8692, Z -8.0000, A 0.000, B 0.000, C 0.000 }
gfCNCPoint6[10416] = {X 533.9633, Y 7.8692, Z -8.0000, A 0.000, B 0.000, C 0.000 }
gfCNCPoint6[10417] = {X 533.9633, Y 3.8692, Z -8.0000, A 0.000, B 0.000, C 0.000 }
gfCNCPoint6[10418] = {X 533.9633, Y 7.9492, Z -8.0000, A 0.000, B 0.000, C 0.000 }
gfCNCPoint6[10419] = {X 543.7510, Y 7.9492, Z -8.0000, A 0.000, B 0.000, C 0.000 }
gfCNCPoint6[10420] = {X 544.7135, Y 8.0330, Z -8.0000, A 0.000, B 0.000, C 0.000 }
gfCNCPoint6[10421] = {X 545.6321, Y 8.3322, Z -8.0000, A 0.000, B 0.000, C 0.000 }
gfCNCPoint6[10422] = {X 546.4593, Y 8.8313, Z -8.0000, A 0.000, B 0.000, C 0.000 }
gfCNCPoint6[10423] = {X 547.1521, Y 9.5046, Z -8.0000, A 0.000, B 0.000, C 0.000 }
gfCNCPoint6[10424] = {X 547.6748, Y 10.3171, Z -8.0000, A 0.000, B 0.000, C 0.000 }
gfCNCPoint6[10425] = {X 548.0002, Y 11.2268, Z -8.0000, A 0.000, B 0.000, C 0.000 }
gfCNCPoint6[10426] = {X 548.1114, Y 12.1865, Z -8.0000, A 0.000, B 0.000, C 0.000 }
gfCNCPoint6[10427] = {X 548.1112, Y 13.0217, Z -8.0000, A 0.000, B 0.000, C 0.000 }
gfCNCPoint6[10428] = {X 548.0029, Y 13.9312, Z -8.0000, A 0.000, B 0.000, C 0.000 }
gfCNCPoint6[10429] = {X 547.7018, Y 14.7962, Z -8.0000, A 0.000, B 0.000, C 0.000 }
gfCNCPoint6[10430] = {X 547.2220, Y 15.5764, Z -8.0000, A 0.000, B 0.000, C 0.000 }
gfCNCPoint6[10431] = {X 546.5858, Y 16.2353, Z -8.0000, A 0.000, B 0.000, C 0.000 }
gfCNCPoint6[10432] = {X 546.5853, Y 40.9521, Z -8.0000, A 0.000, B 0.000, C 0.000 }
gfCNCPoint6[10433] = {X 546.6354, Y 40.9935, Z -8.0000, A 0.000, B 0.000, C 0.000 }
gfCNCPoint6[10434] = {X 547.2530, Y 41.6509, Z -8.0000, A 0.000, B 0.000, C 0.000 }
gfCNCPoint6[10435] = {X 547.7175, Y 42.4240, Z -8.0000, A 0.000, B 0.000, C 0.000 }
gfCNCPoint6[10436] = {X 548.0080, Y 43.2779, Z -8.0000, A 0.000, B 0.000, C 0.000 }
gfCNCPoint6[10437] = {X 548.1113, Y 44.1740, Z -8.0000, A 0.000, B 0.000, C 0.000 }
gfCNCPoint6[10438] = {X 548.1114, Y 45.0003, Z -8.0000, A 0.000, B 0.000, C 0.000 }
gfCNCPoint6[10439] = {X 548.0001, Y 45.9600, Z -8.0000, A 0.000, B 0.000, C 0.000 }
gfCNCPoint6[10440] = {X 547.6747, Y 46.8696, Z -8.0000, A 0.000, B 0.000, C 0.000 }
gfCNCPoint6[10441] = {X 547.1520, Y 47.6821, Z -8.0000, A 0.000, B 0.000, C 0.000 }
gfCNCPoint6[10442] = {X 546.4592, Y 48.3553, Z -8.0000, A 0.000, B 0.000, C 0.000 }
gfCNCPoint6[10443] = {X 545.6320, Y 48.8544, Z -8.0000, A 0.000, B 0.000, C 0.000 }
gfCNCPoint6[10444] = {X 544.7134, Y 49.1536, Z -8.0000, A 0.000, B 0.000, C 0.000 }
gfCNCPoint6[10445] = {X 543.7510, Y 49.2373, Z -8.0000, A 0.000, B 0.000, C 0.000 }
gfCNCPoint6[10446] = {X 524.0042, Y 49.2376, Z -8.0000, A 0.000, B 0.000, C 0.000 }
gfCNCPoint6[10447] = {X 523.4673, Y 49.8707, Z -8.0000, A 0.000, B 0.000, C 0.000 }
gfCNCPoint6[10448] = {X 522.8210, Y 50.3917, Z -8.0000, A 0.000, B 0.000, C 0.000 }
gfCNCPoint6[10449] = {X 522.0882, Y 50.7818, Z -8.0000, A 0.000, B 0.000, C 0.000 }
gfCNCPoint6[10450] = {X 521.2952, Y 51.0272, Z -8.0000, A 0.000, B 0.000, C 0.000 }
gfCNCPoint6[10451] = {X 520.4701, Y 51.1191, Z -8.0000, A 0.000, B 0.000, C 0.000 }
gfCNCPoint6[10452] = {X 519.7998, Y 51.1191, Z -8.0000, A 0.000, B 0.000, C 0.000 }
gfCNCPoint6[10453] = {X 518.8563, Y 51.0128, Z -8.0000, A 0.000, B 0.000, C 0.000 }
gfCNCPoint6[10454] = {X 517.9601, Y 50.6992, Z -8.0000, A 0.000, B 0.000, C 0.000 }
gfCNCPoint6[10455] = {X 517.1562, Y 50.1941, Z -8.0000, A 0.000, B 0.000, C 0.000 }
gfCNCPoint6[10456] = {X 516.4848, Y 49.5227, Z -8.0000, A 0.000, B 0.000, C 0.000 }
gfCNCPoint6[10457] = {X 515.9797, Y 48.7188, Z -8.0000, A 0.000, B 0.000, C 0.000 }
gfCNCPoint6[10458] = {X 515.6661, Y 47.8226, Z -8.0000, A 0.000, B 0.000, C 0.000 }
gfCNCPoint6[10459] = {X 515.5598, Y 46.8791, Z -8.0000, A 0.000, B 0.000, C 0.000 }
gfCNCPoint6[10460] = {X 515.5598, Y 39.9011, Z -8.0000, A 0.000, B 0.000, C 0.000 }
gfCNCPoint6[10461] = {X 515.6649, Y 38.9628, Z -8.0000, A 0.000, B 0.000, C 0.000 }
gfCNCPoint6[10462] = {X 515.9751, Y 38.0710, Z -8.0000, A 0.000, B 0.000, C 0.000 }
gfCNCPoint6[10463] = {X 516.4749, Y 37.2700, Z -8.0000, A 0.000, B 0.000, C 0.000 }
gfCNCPoint6[10464] = {X 517.1395, Y 36.5995, Z -8.0000, A 0.000, B 0.000, C 0.000 }
gfCNCPoint6[10465] = {X 517.9361, Y 36.0926, Z -8.0000, A 0.000, B 0.000, C 0.000 }
gfCNCPoint6[10466] = {X 518.8251, Y 35.7746, Z -8.0000, A 0.000, B 0.000, C 0.000 }
gfCNCPoint6[10467] = {X 519.7624, Y 35.6613, Z -8.0000, A 0.000, B 0.000, C 0.000 }
gfCNCPoint6[10468] = {X 520.5258, Y 35.6615, Z -8.0000, A 0.000, B 0.000, C 0.000 }
gfCNCPoint6[10469] = {X 521.3450, Y 35.7528, Z -8.0000, A 0.000, B 0.000, C 0.000 }
gfCNCPoint6[10470] = {X 522.1312, Y 36.0008, Z -8.0000, A 0.000, B 0.000, C 0.000 }
gfCNCPoint6[10471] = {X 522.8544, Y 36.3963, Z -8.0000, A 0.000, B 0.000, C 0.000 }
gfCNCPoint6[10472] = {X 523.4875, Y 36.9243, Z -8.0000, A 0.000, B 0.000, C 0.000 }
gfCNCPoint6[10473] = {X 524.0064, Y 37.5648, Z -8.0000, A 0.000, B 0.000, C 0.000 }
gfCNCPoint6[10474] = {X 534.7119, Y 37.5648, Z -8.0000, A 0.000, B 0.000, C 0.000 }
gfCNCPoint6[10475] = {X 534.7119, Y 33.8864, Z -8.0000, A 0.000, B 0.000, C 0.000 }
gfCNCPoint6[10476] = {X 530.0653, Y 33.8863, Z -8.0000, A 0.000, B 0.000, C 0.000 }
gfCNCPoint6[10477] = {X 530.0413, Y 33.9237, Z -8.0000, A 0.000, B 0.000, C 0.000 }
gfCNCPoint6[10478] = {X 529.5190, Y 34.5552, Z -8.0000, A 0.000, B 0.000, C 0.000 }
gfCNCPoint6[10479] = {X 528.8849, Y 35.0743, Z -8.0000, A 0.000, B 0.000, C 0.000 }
gfCNCPoint6[10480] = {X 528.1628, Y 35.4618, Z -8.0000, A 0.000, B 0.000, C 0.000 }
gfCNCPoint6[10481] = {X 527.3797, Y 35.7031, Z -8.0000, A 0.000, B 0.000, C 0.000 }
gfCNCPoint6[10482] = {X 526.5648, Y 35.7893, Z -8.0000, A 0.000, B 0.000, C 0.000 }
gfCNCPoint6[10483] = {X 525.8868, Y 35.7895, Z -8.0000, A 0.000, B 0.000, C 0.000 }
gfCNCPoint6[10484] = {X 524.9433, Y 35.6831, Z -8.0000, A 0.000, B 0.000, C 0.000 }
gfCNCPoint6[10485] = {X 524.0471, Y 35.3696, Z -8.0000, A 0.000, B 0.000, C 0.000 }
gfCNCPoint6[10486] = {X 523.2432, Y 34.8644, Z -8.0000, A 0.000, B 0.000, C 0.000 }
gfCNCPoint6[10487] = {X 522.5718, Y 34.1930, Z -8.0000, A 0.000, B 0.000, C 0.000 }
gfCNCPoint6[10488] = {X 522.0666, Y 33.3891, Z -8.0000, A 0.000, B 0.000, C 0.000 }
gfCNCPoint6[10489] = {X 521.7531, Y 32.4929, Z -8.0000, A 0.000, B 0.000, C 0.000 }
gfCNCPoint6[10490] = {X 521.6468, Y 31.5495, Z -8.0000, A 0.000, B 0.000, C 0.000 }
gfCNCPoint6[10491] = {X 521.6468, Y 24.5714, Z -8.0000, A 0.000, B 0.000, C 0.000 }
gfCNCPoint6[10492] = {X 521.7519, Y 23.6330, Z -8.0000, A 0.000, B 0.000, C 0.000 }
gfCNCPoint6[10493] = {X 522.0622, Y 22.7411, Z -8.0000, A 0.000, B 0.000, C 0.000 }
gfCNCPoint6[10494] = {X 522.5621, Y 21.9400, Z -8.0000, A 0.000, B 0.000, C 0.000 }
gfCNCPoint6[10495] = {X 523.2270, Y 21.2694, Z -8.0000, A 0.000, B 0.000, C 0.000 }
gfCNCPoint6[10496] = {X 524.0238, Y 20.7626, Z -8.0000, A 0.000, B 0.000, C 0.000 }
gfCNCPoint6[10497] = {X 524.9130, Y 20.4448, Z -8.0000, A 0.000, B 0.000, C 0.000 }
gfCNCPoint6[10498] = {X 525.8505, Y 20.3316, Z -8.0000, A 0.000, B 0.000, C 0.000 }
gfCNCPoint6[10499] = {X 526.5687, Y 20.3316, Z -8.0000, A 0.000, B 0.000, C 0.000 }
gfCNCPoint6[10500] = {X 527.3865, Y 20.4192, Z -8.0000, A 0.000, B 0.000, C 0.000 }
gfCNCPoint6[10501] = {X 528.1719, Y 20.6629, Z -8.0000, A 0.000, B 0.000, C 0.000 }
gfCNCPoint6[10502] = {X 528.8956, Y 21.0537, Z -8.0000, A 0.000, B 0.000, C 0.000 }
gfCNCPoint6[10503] = {X 529.5302, Y 21.5769, Z -8.0000, A 0.000, B 0.000, C 0.000 }
gfCNCPoint6[10504] = {X 530.0518, Y 22.2127, Z -8.0000, A 0.000, B 0.000, C 0.000 }
gfCNCPoint6[10505] = {X 534.7119, Y 22.2127, Z -8.0000, A 0.000, B 0.000, C 0.000 }
gfCNCPoint6[10506] = {X 534.7119, Y 19.6228, Z -8.0000, A 0.000, B 0.000, C 0.000 }
gfCNCPoint6[10507] = {X 524.1484, Y 19.6228, Z -8.0000, A 0.000, B 0.000, C 0.000 }
gfCNCPoint6[10508] = {X 524.1250, Y 19.6580, Z -8.0000, A 0.000, B 0.000, C 0.000 }
gfCNCPoint6[10509] = {X 523.6024, Y 20.2903, Z -8.0000, A 0.000, B 0.000, C 0.000 }
gfCNCPoint6[10510] = {X 522.9679, Y 20.8102, Z -8.0000, A 0.000, B 0.000, C 0.000 }
gfCNCPoint6[10511] = {X 522.2451, Y 21.1981, Z -8.0000, A 0.000, B 0.000, C 0.000 }
gfCNCPoint6[10512] = {X 521.4611, Y 21.4396, Z -8.0000, A 0.000, B 0.000, C 0.000 }
gfCNCPoint6[10513] = {X 520.6453, Y 21.5256, Z -8.0000, A 0.000, B 0.000, C 0.000 }
gfCNCPoint6[10514] = {X 519.9691, Y 21.5257, Z -8.0000, A 0.000, B 0.000, C 0.000 }
gfCNCPoint6[10515] = {X 519.0256, Y 21.4194, Z -8.0000, A 0.000, B 0.000, C 0.000 }
gfCNCPoint6[10516] = {X 518.1294, Y 21.1058, Z -8.0000, A 0.000, B 0.000, C 0.000 }
gfCNCPoint6[10517] = {X 517.3255, Y 20.6007, Z -8.0000, A 0.000, B 0.000, C 0.000 }
gfCNCPoint6[10518] = {X 516.6541, Y 19.9293, Z -8.0000, A 0.000, B 0.000, C 0.000 }
gfCNCPoint6[10519] = {X 516.1490, Y 19.1254, Z -8.0000, A 0.000, B 0.000, C 0.000 }
gfCNCPoint6[10520] = {X 515.8354, Y 18.2292, Z -8.0000, A 0.000, B 0.000, C 0.000 }
gfCNCPoint6[10521] = {X 515.7291, Y 17.2857, Z -8.0000, A 0.000, B 0.000, C 0.000 }
gfCNCPoint6[10522] = {X 515.7291, Y 10.3077, Z -8.0000, A 0.000, B 0.000, C 0.000 }
gfCNCPoint6[10523] = {X 515.8342, Y 9.3696, Z -8.0000, A 0.000, B 0.000, C 0.000 }
gfCNCPoint6[10524] = {X 516.1442, Y 8.4780, Z -8.0000, A 0.000, B 0.000, C 0.000 }
gfCNCPoint6[10525] = {X 516.6438, Y 7.6771, Z -8.0000, A 0.000, B 0.000, C 0.000 }
gfCNCPoint6[10526] = {X 517.3082, Y 7.0066, Z -8.0000, A 0.000, B 0.000, C 0.000 }
gfCNCPoint6[10527] = {X 518.1045, Y 6.4997, Z -8.0000, A 0.000, B 0.000, C 0.000 }
gfCNCPoint6[10528] = {X 518.9932, Y 6.1815, Z -8.0000, A 0.000, B 0.000, C 0.000 }
gfCNCPoint6[10529] = {X 519.9303, Y 6.0679, Z -8.0000, A 0.000, B 0.000, C 0.000 }
gfCNCPoint6[10530] = {X 520.6494, Y 6.0679, Z -8.0000, A 0.000, B 0.000, C 0.000 }
gfCNCPoint6[10531] = {X 521.4676, Y 6.1552, Z -8.0000, A 0.000, B 0.000, C 0.000 }
gfCNCPoint6[10532] = {X 522.2535, Y 6.3988, Z -8.0000, A 0.000, B 0.000, C 0.000 }
gfCNCPoint6[10533] = {X 522.9775, Y 6.7897, Z -8.0000, A 0.000, B 0.000, C 0.000 }
gfCNCPoint6[10534] = {X 523.6124, Y 7.3131, Z -8.0000, A 0.000, B 0.000, C 0.000 }
gfCNCPoint6[10535] = {X 524.1343, Y 7.9492, Z -8.0000, A 0.000, B 0.000, C 0.000 }
gfCNCPoint6[10536] = {X 533.9633, Y 7.9492, Z -8.0000, A 0.000, B 0.000, C 0.000 }
gfCNCPoint6[10537] = {X 533.9633, Y 3.9492, Z -8.0000, A 0.000, B 0.000, C 0.000 }
gfCNCPoint6[10538] = {X 533.9633, Y 8.0292, Z -8.0000, A 0.000, B 0.000, C 0.000 }
gfCNCPoint6[10539] = {X 543.7521, Y 8.0292, Z -8.0000, A 0.000, B 0.000, C 0.000 }
gfCNCPoint6[10540] = {X 544.6966, Y 8.1112, Z -8.0000, A 0.000, B 0.000, C 0.000 }
gfCNCPoint6[10541] = {X 545.5981, Y 8.4046, Z -8.0000, A 0.000, B 0.000, C 0.000 }
gfCNCPoint6[10542] = {X 546.4099, Y 8.8943, Z -8.0000, A 0.000, B 0.000, C 0.000 }
gfCNCPoint6[10543] = {X 547.0899, Y 9.5549, Z -8.0000, A 0.000, B 0.000, C 0.000 }
gfCNCPoint6[10544] = {X 547.6029, Y 10.3522, Z -8.0000, A 0.000, B 0.000, C 0.000 }
gfCNCPoint6[10545] = {X 547.9222, Y 11.2449, Z -8.0000, A 0.000, B 0.000, C 0.000 }
gfCNCPoint6[10546] = {X 548.0314, Y 12.1866, Z -8.0000, A 0.000, B 0.000, C 0.000 }
gfCNCPoint6[10547] = {X 548.0312, Y 13.0208, Z -8.0000, A 0.000, B 0.000, C 0.000 }
gfCNCPoint6[10548] = {X 547.9228, Y 13.9223, Z -8.0000, A 0.000, B 0.000, C 0.000 }
gfCNCPoint6[10549] = {X 547.6215, Y 14.7787, Z -8.0000, A 0.000, B 0.000, C 0.000 }
gfCNCPoint6[10550] = {X 547.1415, Y 15.5494, Z -8.0000, A 0.000, B 0.000, C 0.000 }
gfCNCPoint6[10551] = {X 546.5058, Y 16.1976, Z -8.0000, A 0.000, B 0.000, C 0.000 }
gfCNCPoint6[10552] = {X 546.5053, Y 40.9898, Z -8.0000, A 0.000, B 0.000, C 0.000 }
gfCNCPoint6[10553] = {X 546.5839, Y 41.0547, Z -8.0000, A 0.000, B 0.000, C 0.000 }
gfCNCPoint6[10554] = {X 547.1895, Y 41.6996, Z -8.0000, A 0.000, B 0.000, C 0.000 }
gfCNCPoint6[10555] = {X 547.6451, Y 42.4581, Z -8.0000, A 0.000, B 0.000, C 0.000 }
gfCNCPoint6[10556] = {X 547.9300, Y 43.2957, Z -8.0000, A 0.000, B 0.000, C 0.000 }
gfCNCPoint6[10557] = {X 548.0313, Y 44.1746, Z -8.0000, A 0.000, B 0.000, C 0.000 }
gfCNCPoint6[10558] = {X 548.0314, Y 45.0002, Z -8.0000, A 0.000, B 0.000, C 0.000 }
gfCNCPoint6[10559] = {X 547.9222, Y 45.9419, Z -8.0000, A 0.000, B 0.000, C 0.000 }
gfCNCPoint6[10560] = {X 547.6028, Y 46.8345, Z -8.0000, A 0.000, B 0.000, C 0.000 }
gfCNCPoint6[10561] = {X 547.0898, Y 47.6318, Z -8.0000, A 0.000, B 0.000, C 0.000 }
gfCNCPoint6[10562] = {X 546.4098, Y 48.2923, Z -8.0000, A 0.000, B 0.000, C 0.000 }
gfCNCPoint6[10563] = {X 545.5981, Y 48.7820, Z -8.0000, A 0.000, B 0.000, C 0.000 }
gfCNCPoint6[10564] = {X 544.6966, Y 49.0754, Z -8.0000, A 0.000, B 0.000, C 0.000 }
gfCNCPoint6[10565] = {X 543.7521, Y 49.1573, Z -8.0000, A 0.000, B 0.000, C 0.000 }
gfCNCPoint6[10566] = {X 523.9622, Y 49.1576, Z -8.0000, A 0.000, B 0.000, C 0.000 }
gfCNCPoint6[10567] = {X 523.4353, Y 49.7900, Z -8.0000, A 0.000, B 0.000, C 0.000 }
gfCNCPoint6[10568] = {X 522.7979, Y 50.3110, Z -8.0000, A 0.000, B 0.000, C 0.000 }
gfCNCPoint6[10569] = {X 522.0732, Y 50.7014, Z -8.0000, A 0.000, B 0.000, C 0.000 }
gfCNCPoint6[10570] = {X 521.2875, Y 50.9471, Z -8.0000, A 0.000, B 0.000, C 0.000 }
gfCNCPoint6[10571] = {X 520.4695, Y 51.0391, Z -8.0000, A 0.000, B 0.000, C 0.000 }
gfCNCPoint6[10572] = {X 519.7998, Y 51.0391, Z -8.0000, A 0.000, B 0.000, C 0.000 }
gfCNCPoint6[10573] = {X 518.8741, Y 50.9348, Z -8.0000, A 0.000, B 0.000, C 0.000 }
gfCNCPoint6[10574] = {X 517.9948, Y 50.6272, Z -8.0000, A 0.000, B 0.000, C 0.000 }
gfCNCPoint6[10575] = {X 517.2061, Y 50.1315, Z -8.0000, A 0.000, B 0.000, C 0.000 }
gfCNCPoint6[10576] = {X 516.5474, Y 49.4728, Z -8.0000, A 0.000, B 0.000, C 0.000 }
gfCNCPoint6[10577] = {X 516.0517, Y 48.6841, Z -8.0000, A 0.000, B 0.000, C 0.000 }
gfCNCPoint6[10578] = {X 515.7441, Y 47.8048, Z -8.0000, A 0.000, B 0.000, C 0.000 }
gfCNCPoint6[10579] = {X 515.6398, Y 46.8791, Z -8.0000, A 0.000, B 0.000, C 0.000 }
gfCNCPoint6[10580] = {X 515.6398, Y 39.9011, Z -8.0000, A 0.000, B 0.000, C 0.000 }
gfCNCPoint6[10581] = {X 515.7429, Y 38.9805, Z -8.0000, A 0.000, B 0.000, C 0.000 }
gfCNCPoint6[10582] = {X 516.0472, Y 38.1056, Z -8.0000, A 0.000, B 0.000, C 0.000 }
gfCNCPoint6[10583] = {X 516.5376, Y 37.3197, Z -8.0000, A 0.000, B 0.000, C 0.000 }
gfCNCPoint6[10584] = {X 517.1897, Y 36.6618, Z -8.0000, A 0.000, B 0.000, C 0.000 }
gfCNCPoint6[10585] = {X 517.9713, Y 36.1645, Z -8.0000, A 0.000, B 0.000, C 0.000 }
gfCNCPoint6[10586] = {X 518.8435, Y 35.8525, Z -8.0000, A 0.000, B 0.000, C 0.000 }
gfCNCPoint6[10587] = {X 519.7631, Y 35.7413, Z -8.0000, A 0.000, B 0.000, C 0.000 }
gfCNCPoint6[10588] = {X 520.5247, Y 35.7415, Z -8.0000, A 0.000, B 0.000, C 0.000 }
gfCNCPoint6[10589] = {X 521.3369, Y 35.8328, Z -8.0000, A 0.000, B 0.000, C 0.000 }
gfCNCPoint6[10590] = {X 522.1156, Y 36.0812, Z -8.0000, A 0.000, B 0.000, C 0.000 }
gfCNCPoint6[10591] = {X 522.8306, Y 36.4770, Z -8.0000, A 0.000, B 0.000, C 0.000 }
gfCNCPoint6[10592] = {X 523.4545, Y 37.0050, Z -8.0000, A 0.000, B 0.000, C 0.000 }
gfCNCPoint6[10593] = {X 523.9631, Y 37.6448, Z -8.0000, A 0.000, B 0.000, C 0.000 }
gfCNCPoint6[10594] = {X 534.7919, Y 37.6448, Z -8.0000, A 0.000, B 0.000, C 0.000 }
gfCNCPoint6[10595] = {X 534.7919, Y 33.8064, Z -8.0000, A 0.000, B 0.000, C 0.000 }
gfCNCPoint6[10596] = {X 530.0215, Y 33.8063, Z -8.0000, A 0.000, B 0.000, C 0.000 }
gfCNCPoint6[10597] = {X 529.9745, Y 33.8797, Z -8.0000, A 0.000, B 0.000, C 0.000 }
gfCNCPoint6[10598] = {X 529.4620, Y 34.4990, Z -8.0000, A 0.000, B 0.000, C 0.000 }
gfCNCPoint6[10599] = {X 528.8400, Y 35.0081, Z -8.0000, A 0.000, B 0.000, C 0.000 }
gfCNCPoint6[10600] = {X 528.1316, Y 35.3881, Z -8.0000, A 0.000, B 0.000, C 0.000 }
gfCNCPoint6[10601] = {X 527.3634, Y 35.6248, Z -8.0000, A 0.000, B 0.000, C 0.000 }
gfCNCPoint6[10602] = {X 526.5641, Y 35.7093, Z -8.0000, A 0.000, B 0.000, C 0.000 }
gfCNCPoint6[10603] = {X 525.8868, Y 35.7095, Z -8.0000, A 0.000, B 0.000, C 0.000 }
gfCNCPoint6[10604] = {X 524.9611, Y 35.6052, Z -8.0000, A 0.000, B 0.000, C 0.000 }
gfCNCPoint6[10605] = {X 524.0818, Y 35.2975, Z -8.0000, A 0.000, B 0.000, C 0.000 }
gfCNCPoint6[10606] = {X 523.2930, Y 34.8019, Z -8.0000, A 0.000, B 0.000, C 0.000 }
gfCNCPoint6[10607] = {X 522.6343, Y 34.1432, Z -8.0000, A 0.000, B 0.000, C 0.000 }
gfCNCPoint6[10608] = {X 522.1387, Y 33.3544, Z -8.0000, A 0.000, B 0.000, C 0.000 }
gfCNCPoint6[10609] = {X 521.8311, Y 32.4751, Z -8.0000, A 0.000, B 0.000, C 0.000 }
gfCNCPoint6[10610] = {X 521.7268, Y 31.5495, Z -8.0000, A 0.000, B 0.000, C 0.000 }
gfCNCPoint6[10611] = {X 521.7268, Y 24.5714, Z -8.0000, A 0.000, B 0.000, C 0.000 }
gfCNCPoint6[10612] = {X 521.8299, Y 23.6507, Z -8.0000, A 0.000, B 0.000, C 0.000 }
gfCNCPoint6[10613] = {X 522.1343, Y 22.7756, Z -8.0000, A 0.000, B 0.000, C 0.000 }
gfCNCPoint6[10614] = {X 522.6248, Y 21.9897, Z -8.0000, A 0.000, B 0.000, C 0.000 }
gfCNCPoint6[10615] = {X 523.2772, Y 21.3317, Z -8.0000, A 0.000, B 0.000, C 0.000 }
gfCNCPoint6[10616] = {X 524.0589, Y 20.8345, Z -8.0000, A 0.000, B 0.000, C 0.000 }
gfCNCPoint6[10617] = {X 524.9313, Y 20.5226, Z -8.0000, A 0.000, B 0.000, C 0.000 }
gfCNCPoint6[10618] = {X 525.8511, Y 20.4116, Z -8.0000, A 0.000, B 0.000, C 0.000 }
gfCNCPoint6[10619] = {X 526.5679, Y 20.4116, Z -8.0000, A 0.000, B 0.000, C 0.000 }
gfCNCPoint6[10620] = {X 527.3786, Y 20.4992, Z -8.0000, A 0.000, B 0.000, C 0.000 }
gfCNCPoint6[10621] = {X 528.1566, Y 20.7433, Z -8.0000, A 0.000, B 0.000, C 0.000 }
gfCNCPoint6[10622] = {X 528.8721, Y 21.1344, Z -8.0000, A 0.000, B 0.000, C 0.000 }
gfCNCPoint6[10623] = {X 529.4975, Y 21.6576, Z -8.0000, A 0.000, B 0.000, C 0.000 }
gfCNCPoint6[10624] = {X 530.0088, Y 22.2927, Z -8.0000, A 0.000, B 0.000, C 0.000 }
gfCNCPoint6[10625] = {X 534.7919, Y 22.2927, Z -8.0000, A 0.000, B 0.000, C 0.000 }
gfCNCPoint6[10626] = {X 534.7919, Y 19.5428, Z -8.0000, A 0.000, B 0.000, C 0.000 }
gfCNCPoint6[10627] = {X 524.1047, Y 19.5428, Z -8.0000, A 0.000, B 0.000, C 0.000 }
gfCNCPoint6[10628] = {X 524.0760, Y 19.5875, Z -8.0000, A 0.000, B 0.000, C 0.000 }
gfCNCPoint6[10629] = {X 523.5635, Y 20.2161, Z -8.0000, A 0.000, B 0.000, C 0.000 }
gfCNCPoint6[10630] = {X 522.9388, Y 20.7333, Z -8.0000, A 0.000, B 0.000, C 0.000 }
gfCNCPoint6[10631] = {X 522.2257, Y 21.1195, Z -8.0000, A 0.000, B 0.000, C 0.000 }
gfCNCPoint6[10632] = {X 521.4512, Y 21.3599, Z -8.0000, A 0.000, B 0.000, C 0.000 }
gfCNCPoint6[10633] = {X 520.6447, Y 21.4456, Z -8.0000, A 0.000, B 0.000, C 0.000 }
gfCNCPoint6[10634] = {X 519.9691, Y 21.4457, Z -8.0000, A 0.000, B 0.000, C 0.000 }
gfCNCPoint6[10635] = {X 519.0434, Y 21.3414, Z -8.0000, A 0.000, B 0.000, C 0.000 }
gfCNCPoint6[10636] = {X 518.1641, Y 21.0337, Z -8.0000, A 0.000, B 0.000, C 0.000 }
gfCNCPoint6[10637] = {X 517.3754, Y 20.5381, Z -8.0000, A 0.000, B 0.000, C 0.000 }
gfCNCPoint6[10638] = {X 516.7167, Y 19.8794, Z -8.0000, A 0.000, B 0.000, C 0.000 }
gfCNCPoint6[10639] = {X 516.2211, Y 19.0907, Z -8.0000, A 0.000, B 0.000, C 0.000 }
gfCNCPoint6[10640] = {X 515.9134, Y 18.2114, Z -8.0000, A 0.000, B 0.000, C 0.000 }
gfCNCPoint6[10641] = {X 515.8091, Y 17.2857, Z -8.0000, A 0.000, B 0.000, C 0.000 }
gfCNCPoint6[10642] = {X 515.8091, Y 10.3077, Z -8.0000, A 0.000, B 0.000, C 0.000 }
gfCNCPoint6[10643] = {X 515.9122, Y 9.3873, Z -8.0000, A 0.000, B 0.000, C 0.000 }
gfCNCPoint6[10644] = {X 516.2164, Y 8.5125, Z -8.0000, A 0.000, B 0.000, C 0.000 }
gfCNCPoint6[10645] = {X 516.7065, Y 7.7267, Z -8.0000, A 0.000, B 0.000, C 0.000 }
gfCNCPoint6[10646] = {X 517.3584, Y 7.0689, Z -8.0000, A 0.000, B 0.000, C 0.000 }
gfCNCPoint6[10647] = {X 518.1397, Y 6.5715, Z -8.0000, A 0.000, B 0.000, C 0.000 }
gfCNCPoint6[10648] = {X 519.0117, Y 6.2594, Z -8.0000, A 0.000, B 0.000, C 0.000 }
gfCNCPoint6[10649] = {X 519.9311, Y 6.1479, Z -8.0000, A 0.000, B 0.000, C 0.000 }
gfCNCPoint6[10650] = {X 520.6487, Y 6.1479, Z -8.0000, A 0.000, B 0.000, C 0.000 }
gfCNCPoint6[10651] = {X 521.4598, Y 6.2352, Z -8.0000, A 0.000, B 0.000, C 0.000 }
gfCNCPoint6[10652] = {X 522.2382, Y 6.4792, Z -8.0000, A 0.000, B 0.000, C 0.000 }
gfCNCPoint6[10653] = {X 522.9540, Y 6.8704, Z -8.0000, A 0.000, B 0.000, C 0.000 }
gfCNCPoint6[10654] = {X 523.5798, Y 7.3938, Z -8.0000, A 0.000, B 0.000, C 0.000 }
gfCNCPoint6[10655] = {X 524.0913, Y 8.0292, Z -8.0000, A 0.000, B 0.000, C 0.000 }
gfCNCPoint6[10656] = {X 533.9633, Y 8.0292, Z -8.0000, A 0.000, B 0.000, C 0.000 }
gfCNCPoint6[10657] = {X 533.9633, Y 4.0292, Z -8.0000, A 0.000, B 0.000, C 0.000 }
gfCNCPoint6[10658] = {X 533.9633, Y 8.1092, Z -8.0000, A 0.000, B 0.000, C 0.000 }
gfCNCPoint6[10659] = {X 543.7532, Y 8.1092, Z -8.0000, A 0.000, B 0.000, C 0.000 }
gfCNCPoint6[10660] = {X 544.6798, Y 8.1894, Z -8.0000, A 0.000, B 0.000, C 0.000 }
gfCNCPoint6[10661] = {X 545.5642, Y 8.4770, Z -8.0000, A 0.000, B 0.000, C 0.000 }
gfCNCPoint6[10662] = {X 546.3606, Y 8.9573, Z -8.0000, A 0.000, B 0.000, C 0.000 }
gfCNCPoint6[10663] = {X 547.0277, Y 9.6052, Z -8.0000, A 0.000, B 0.000, C 0.000 }
gfCNCPoint6[10664] = {X 547.5310, Y 10.3873, Z -8.0000, A 0.000, B 0.000, C 0.000 }
gfCNCPoint6[10665] = {X 547.8443, Y 11.2629, Z -8.0000, A 0.000, B 0.000, C 0.000 }
gfCNCPoint6[10666] = {X 547.9514, Y 12.1867, Z -8.0000, A 0.000, B 0.000, C 0.000 }
gfCNCPoint6[10667] = {X 547.9512, Y 13.0200, Z -8.0000, A 0.000, B 0.000, C 0.000 }
gfCNCPoint6[10668] = {X 547.8428, Y 13.9133, Z -8.0000, A 0.000, B 0.000, C 0.000 }
gfCNCPoint6[10669] = {X 547.5412, Y 14.7611, Z -8.0000, A 0.000, B 0.000, C 0.000 }
gfCNCPoint6[10670] = {X 547.0611, Y 15.5222, Z -8.0000, A 0.000, B 0.000, C 0.000 }
gfCNCPoint6[10671] = {X 546.4258, Y 16.1595, Z -8.0000, A 0.000, B 0.000, C 0.000 }
gfCNCPoint6[10672] = {X 546.4253, Y 41.0275, Z -8.0000, A 0.000, B 0.000, C 0.000 }
gfCNCPoint6[10673] = {X 546.5323, Y 41.1159, Z -8.0000, A 0.000, B 0.000, C 0.000 }
gfCNCPoint6[10674] = {X 547.1261, Y 41.7484, Z -8.0000, A 0.000, B 0.000, C 0.000 }
gfCNCPoint6[10675] = {X 547.5727, Y 42.4921, Z -8.0000, A 0.000, B 0.000, C 0.000 }
gfCNCPoint6[10676] = {X 547.8520, Y 43.3134, Z -8.0000, A 0.000, B 0.000, C 0.000 }
gfCNCPoint6[10677] = {X 547.9513, Y 44.1753, Z -8.0000, A 0.000, B 0.000, C 0.000 }
gfCNCPoint6[10678] = {X 547.9514, Y 45.0001, Z -8.0000, A 0.000, B 0.000, C 0.000 }
gfCNCPoint6[10679] = {X 547.8443, Y 45.9239, Z -8.0000, A 0.000, B 0.000, C 0.000 }
gfCNCPoint6[10680] = {X 547.5309, Y 46.7995, Z -8.0000, A 0.000, B 0.000, C 0.000 }
gfCNCPoint6[10681] = {X 547.0276, Y 47.5815, Z -8.0000, A 0.000, B 0.000, C 0.000 }
gfCNCPoint6[10682] = {X 546.3605, Y 48.2294, Z -8.0000, A 0.000, B 0.000, C 0.000 }
gfCNCPoint6[10683] = {X 545.5641, Y 48.7095, Z -8.0000, A 0.000, B 0.000, C 0.000 }
gfCNCPoint6[10684] = {X 544.6797, Y 48.9972, Z -8.0000, A 0.000, B 0.000, C 0.000 }
gfCNCPoint6[10685] = {X 543.7532, Y 49.0773, Z -8.0000, A 0.000, B 0.000, C 0.000 }
gfCNCPoint6[10686] = {X 523.9197, Y 49.0776, Z -8.0000, A 0.000, B 0.000, C 0.000 }
gfCNCPoint6[10687] = {X 523.4029, Y 49.7093, Z -8.0000, A 0.000, B 0.000, C 0.000 }
gfCNCPoint6[10688] = {X 522.7746, Y 50.2302, Z -8.0000, A 0.000, B 0.000, C 0.000 }
gfCNCPoint6[10689] = {X 522.0580, Y 50.6209, Z -8.0000, A 0.000, B 0.000, C 0.000 }
gfCNCPoint6[10690] = {X 521.2798, Y 50.8670, Z -8.0000, A 0.000, B 0.000, C 0.000 }
gfCNCPoint6[10691] = {X 520.4688, Y 50.9591, Z -8.0000, A 0.000, B 0.000, C 0.000 }
gfCNCPoint6[10692] = {X 519.7998, Y 50.9591, Z -8.0000, A 0.000, B 0.000, C 0.000 }
gfCNCPoint6[10693] = {X 518.8919, Y 50.8568, Z -8.0000, A 0.000, B 0.000, C 0.000 }
gfCNCPoint6[10694] = {X 518.0295, Y 50.5551, Z -8.0000, A 0.000, B 0.000, C 0.000 }
gfCNCPoint6[10695] = {X 517.2559, Y 50.0690, Z -8.0000, A 0.000, B 0.000, C 0.000 }
gfCNCPoint6[10696] = {X 516.6099, Y 49.4230, Z -8.0000, A 0.000, B 0.000, C 0.000 }
gfCNCPoint6[10697] = {X 516.1238, Y 48.6494, Z -8.0000, A 0.000, B 0.000, C 0.000 }
gfCNCPoint6[10698] = {X 515.8221, Y 47.7870, Z -8.0000, A 0.000, B 0.000, C 0.000 }
gfCNCPoint6[10699] = {X 515.7198, Y 46.8791, Z -8.0000, A 0.000, B 0.000, C 0.000 }
gfCNCPoint6[10700] = {X 515.7198, Y 39.9011, Z -8.0000, A 0.000, B 0.000, C 0.000 }
gfCNCPoint6[10701] = {X 515.8209, Y 38.9982, Z -8.0000, A 0.000, B 0.000, C 0.000 }
gfCNCPoint6[10702] = {X 516.1194, Y 38.1401, Z -8.0000, A 0.000, B 0.000, C 0.000 }
gfCNCPoint6[10703] = {X 516.6003, Y 37.3693, Z -8.0000, A 0.000, B 0.000, C 0.000 }
gfCNCPoint6[10704] = {X 517.2399, Y 36.7241, Z -8.0000, A 0.000, B 0.000, C 0.000 }
gfCNCPoint6[10705] = {X 518.0064, Y 36.2364, Z -8.0000, A 0.000, B 0.000, C 0.000 }
gfCNCPoint6[10706] = {X 518.8619, Y 35.9304, Z -8.0000, A 0.000, B 0.000, C 0.000 }
gfCNCPoint6[10707] = {X 519.7638, Y 35.8213, Z -8.0000, A 0.000, B 0.000, C 0.000 }
gfCNCPoint6[10708] = {X 520.5236, Y 35.8215, Z -8.0000, A 0.000, B 0.000, C 0.000 }
gfCNCPoint6[10709] = {X 521.3287, Y 35.9129, Z -8.0000, A 0.000, B 0.000, C 0.000 }
gfCNCPoint6[10710] = {X 522.0998, Y 36.1616, Z -8.0000, A 0.000, B 0.000, C 0.000 }
gfCNCPoint6[10711] = {X 522.8066, Y 36.5577, Z -8.0000, A 0.000, B 0.000, C 0.000 }
gfCNCPoint6[10712] = {X 523.4212, Y 37.0857, Z -8.0000, A 0.000, B 0.000, C 0.000 }
gfCNCPoint6[10713] = {X 523.9193, Y 37.7248, Z -8.0000, A 0.000, B 0.000, C 0.000 }
gfCNCPoint6[10714] = {X 534.8719, Y 37.7248, Z -8.0000, A 0.000, B 0.000, C 0.000 }
gfCNCPoint6[10715] = {X 534.8719, Y 33.7264, Z -8.0000, A 0.000, B 0.000, C 0.000 }
gfCNCPoint6[10716] = {X 529.9778, Y 33.7263, Z -8.0000, A 0.000, B 0.000, C 0.000 }
gfCNCPoint6[10717] = {X 529.9071, Y 33.8366, Z -8.0000, A 0.000, B 0.000, C 0.000 }
gfCNCPoint6[10718] = {X 529.2612, Y 34.5790, Z -8.0000, A 0.000, B 0.000, C 0.000 }
gfCNCPoint6[10719] = {X 528.4563, Y 35.1452, Z -8.0000, A 0.000, B 0.000, C 0.000 }
gfCNCPoint6[10720] = {X 527.5392, Y 35.5023, Z -8.0000, A 0.000, B 0.000, C 0.000 }
gfCNCPoint6[10721] = {X 526.5634, Y 35.6293, Z -8.0000, A 0.000, B 0.000, C 0.000 }
gfCNCPoint6[10722] = {X 525.8868, Y 35.6295, Z -8.0000, A 0.000, B 0.000, C 0.000 }
gfCNCPoint6[10723] = {X 524.9789, Y 35.5272, Z -8.0000, A 0.000, B 0.000, C 0.000 }
gfCNCPoint6[10724] = {X 524.1165, Y 35.2254, Z -8.0000, A 0.000, B 0.000, C 0.000 }
gfCNCPoint6[10725] = {X 523.3429, Y 34.7393, Z -8.0000, A 0.000, B 0.000, C 0.000 }
gfCNCPoint6[10726] = {X 522.6969, Y 34.0933, Z -8.0000, A 0.000, B 0.000, C 0.000 }
gfCNCPoint6[10727] = {X 522.2108, Y 33.3197, Z -8.0000, A 0.000, B 0.000, C 0.000 }
gfCNCPoint6[10728] = {X 521.9091, Y 32.4573, Z -8.0000, A 0.000, B 0.000, C 0.000 }
gfCNCPoint6[10729] = {X 521.8068, Y 31.5495, Z -8.0000, A 0.000, B 0.000, C 0.000 }
gfCNCPoint6[10730] = {X 521.8068, Y 24.5714, Z -8.0000, A 0.000, B 0.000, C 0.000 }
gfCNCPoint6[10731] = {X 521.9079, Y 23.6684, Z -8.0000, A 0.000, B 0.000, C 0.000 }
gfCNCPoint6[10732] = {X 522.2065, Y 22.8102, Z -8.0000, A 0.000, B 0.000, C 0.000 }
gfCNCPoint6[10733] = {X 522.6876, Y 22.0393, Z -8.0000, A 0.000, B 0.000, C 0.000 }
gfCNCPoint6[10734] = {X 523.3273, Y 21.3940, Z -8.0000, A 0.000, B 0.000, C 0.000 }
gfCNCPoint6[10735] = {X 524.0941, Y 20.9064, Z -8.0000, A 0.000, B 0.000, C 0.000 }
gfCNCPoint6[10736] = {X 524.9497, Y 20.6005, Z -8.0000, A 0.000, B 0.000, C 0.000 }
gfCNCPoint6[10737] = {X 525.8518, Y 20.4916, Z -8.0000, A 0.000, B 0.000, C 0.000 }
gfCNCPoint6[10738] = {X 526.5672, Y 20.4916, Z -8.0000, A 0.000, B 0.000, C 0.000 }
gfCNCPoint6[10739] = {X 527.3707, Y 20.5793, Z -8.0000, A 0.000, B 0.000, C 0.000 }
gfCNCPoint6[10740] = {X 528.1412, Y 20.8237, Z -8.0000, A 0.000, B 0.000, C 0.000 }
gfCNCPoint6[10741] = {X 528.8483, Y 21.2152, Z -8.0000, A 0.000, B 0.000, C 0.000 }
gfCNCPoint6[10742] = {X 529.4644, Y 21.7384, Z -8.0000, A 0.000, B 0.000, C 0.000 }
gfCNCPoint6[10743] = {X 529.9653, Y 22.3727, Z -8.0000, A 0.000, B 0.000, C 0.000 }
gfCNCPoint6[10744] = {X 534.8719, Y 22.3727, Z -8.0000, A 0.000, B 0.000, C 0.000 }
gfCNCPoint6[10745] = {X 534.8719, Y 19.4628, Z -8.0000, A 0.000, B 0.000, C 0.000 }
gfCNCPoint6[10746] = {X 524.0611, Y 19.4628, Z -8.0000, A 0.000, B 0.000, C 0.000 }
gfCNCPoint6[10747] = {X 524.0087, Y 19.5442, Z -8.0000, A 0.000, B 0.000, C 0.000 }
gfCNCPoint6[10748] = {X 523.5061, Y 20.1604, Z -8.0000, A 0.000, B 0.000, C 0.000 }
gfCNCPoint6[10749] = {X 522.8935, Y 20.6674, Z -8.0000, A 0.000, B 0.000, C 0.000 }
gfCNCPoint6[10750] = {X 522.1942, Y 21.0459, Z -8.0000, A 0.000, B 0.000, C 0.000 }
gfCNCPoint6[10751] = {X 521.4348, Y 21.2816, Z -8.0000, A 0.000, B 0.000, C 0.000 }
gfCNCPoint6[10752] = {X 520.6440, Y 21.3656, Z -8.0000, A 0.000, B 0.000, C 0.000 }
gfCNCPoint6[10753] = {X 519.9691, Y 21.3657, Z -8.0000, A 0.000, B 0.000, C 0.000 }
gfCNCPoint6[10754] = {X 519.0612, Y 21.2634, Z -8.0000, A 0.000, B 0.000, C 0.000 }
gfCNCPoint6[10755] = {X 518.1989, Y 20.9617, Z -8.0000, A 0.000, B 0.000, C 0.000 }
gfCNCPoint6[10756] = {X 517.4253, Y 20.4756, Z -8.0000, A 0.000, B 0.000, C 0.000 }
gfCNCPoint6[10757] = {X 516.7792, Y 19.8296, Z -8.0000, A 0.000, B 0.000, C 0.000 }
gfCNCPoint6[10758] = {X 516.2932, Y 19.0560, Z -8.0000, A 0.000, B 0.000, C 0.000 }
gfCNCPoint6[10759] = {X 515.9914, Y 18.1936, Z -8.0000, A 0.000, B 0.000, C 0.000 }
gfCNCPoint6[10760] = {X 515.8891, Y 17.2857, Z -8.0000, A 0.000, B 0.000, C 0.000 }
gfCNCPoint6[10761] = {X 515.8891, Y 10.3077, Z -8.0000, A 0.000, B 0.000, C 0.000 }
gfCNCPoint6[10762] = {X 515.9902, Y 9.4050, Z -8.0000, A 0.000, B 0.000, C 0.000 }
gfCNCPoint6[10763] = {X 516.2885, Y 8.5471, Z -8.0000, A 0.000, B 0.000, C 0.000 }
gfCNCPoint6[10764] = {X 516.7693, Y 7.7764, Z -8.0000, A 0.000, B 0.000, C 0.000 }
gfCNCPoint6[10765] = {X 517.4086, Y 7.1312, Z -8.0000, A 0.000, B 0.000, C 0.000 }
gfCNCPoint6[10766] = {X 518.1749, Y 6.6434, Z -8.0000, A 0.000, B 0.000, C 0.000 }
gfCNCPoint6[10767] = {X 519.0301, Y 6.3372, Z -8.0000, A 0.000, B 0.000, C 0.000 }
gfCNCPoint6[10768] = {X 519.9318, Y 6.2279, Z -8.0000, A 0.000, B 0.000, C 0.000 }
gfCNCPoint6[10769] = {X 520.6480, Y 6.2279, Z -8.0000, A 0.000, B 0.000, C 0.000 }
gfCNCPoint6[10770] = {X 521.4519, Y 6.3153, Z -8.0000, A 0.000, B 0.000, C 0.000 }
gfCNCPoint6[10771] = {X 522.2227, Y 6.5596, Z -8.0000, A 0.000, B 0.000, C 0.000 }
gfCNCPoint6[10772] = {X 522.9303, Y 6.9512, Z -8.0000, A 0.000, B 0.000, C 0.000 }
gfCNCPoint6[10773] = {X 523.5467, Y 7.4746, Z -8.0000, A 0.000, B 0.000, C 0.000 }
gfCNCPoint6[10774] = {X 524.0478, Y 8.1092, Z -8.0000, A 0.000, B 0.000, C 0.000 }
gfCNCPoint6[10775] = {X 533.9633, Y 8.1092, Z -8.0000, A 0.000, B 0.000, C 0.000 }
gfCNCPoint6[10776] = {X 533.9633, Y 4.1092, Z -8.0000, A 0.000, B 0.000, C 0.000 }
gfCNCPoint6[10777] = {X 533.9633, Y 8.1892, Z -8.0000, A 0.000, B 0.000, C 0.000 }
gfCNCPoint6[10778] = {X 543.7544, Y 8.1892, Z -8.0000, A 0.000, B 0.000, C 0.000 }
gfCNCPoint6[10779] = {X 544.6629, Y 8.2676, Z -8.0000, A 0.000, B 0.000, C 0.000 }
gfCNCPoint6[10780] = {X 545.5302, Y 8.5495, Z -8.0000, A 0.000, B 0.000, C 0.000 }
gfCNCPoint6[10781] = {X 546.3112, Y 9.0202, Z -8.0000, A 0.000, B 0.000, C 0.000 }
gfCNCPoint6[10782] = {X 546.9655, Y 9.6555, Z -8.0000, A 0.000, B 0.000, C 0.000 }
gfCNCPoint6[10783] = {X 547.4591, Y 10.4223, Z -8.0000, A 0.000, B 0.000, C 0.000 }
gfCNCPoint6[10784] = {X 547.7664, Y 11.2810, Z -8.0000, A 0.000, B 0.000, C 0.000 }
gfCNCPoint6[10785] = {X 547.8714, Y 12.1868, Z -8.0000, A 0.000, B 0.000, C 0.000 }
gfCNCPoint6[10786] = {X 547.8712, Y 13.0192, Z -8.0000, A 0.000, B 0.000, C 0.000 }
gfCNCPoint6[10787] = {X 547.7627, Y 13.9043, Z -8.0000, A 0.000, B 0.000, C 0.000 }
gfCNCPoint6[10788] = {X 547.4608, Y 14.7433, Z -8.0000, A 0.000, B 0.000, C 0.000 }
gfCNCPoint6[10789] = {X 546.9806, Y 15.4946, Z -8.0000, A 0.000, B 0.000, C 0.000 }
gfCNCPoint6[10790] = {X 546.3458, Y 16.1209, Z -8.0000, A 0.000, B 0.000, C 0.000 }
gfCNCPoint6[10791] = {X 546.3453, Y 41.0652, Z -8.0000, A 0.000, B 0.000, C 0.000 }
gfCNCPoint6[10792] = {X 546.4840, Y 41.1799, Z -8.0000, A 0.000, B 0.000, C 0.000 }
gfCNCPoint6[10793] = {X 547.0695, Y 41.8062, Z -8.0000, A 0.000, B 0.000, C 0.000 }
gfCNCPoint6[10794] = {X 547.5081, Y 42.5430, Z -8.0000, A 0.000, B 0.000, C 0.000 }
gfCNCPoint6[10795] = {X 547.7795, Y 43.3564, Z -8.0000, A 0.000, B 0.000, C 0.000 }
gfCNCPoint6[10796] = {X 547.8714, Y 44.2089, Z -8.0000, A 0.000, B 0.000, C 0.000 }
gfCNCPoint6[10797] = {X 547.8714, Y 45.0000, Z -8.0000, A 0.000, B 0.000, C 0.000 }
gfCNCPoint6[10798] = {X 547.7663, Y 45.9058, Z -8.0000, A 0.000, B 0.000, C 0.000 }
gfCNCPoint6[10799] = {X 547.4590, Y 46.7644, Z -8.0000, A 0.000, B 0.000, C 0.000 }
gfCNCPoint6[10800] = {X 546.9654, Y 47.5312, Z -8.0000, A 0.000, B 0.000, C 0.000 }
gfCNCPoint6[10801] = {X 546.3112, Y 48.1664, Z -8.0000, A 0.000, B 0.000, C 0.000 }
gfCNCPoint6[10802] = {X 545.5302, Y 48.6371, Z -8.0000, A 0.000, B 0.000, C 0.000 }
gfCNCPoint6[10803] = {X 544.6629, Y 48.9189, Z -8.0000, A 0.000, B 0.000, C 0.000 }
gfCNCPoint6[10804] = {X 543.7544, Y 48.9973, Z -8.0000, A 0.000, B 0.000, C 0.000 }
gfCNCPoint6[10805] = {X 523.8767, Y 48.9976, Z -8.0000, A 0.000, B 0.000, C 0.000 }
gfCNCPoint6[10806] = {X 523.3702, Y 49.6286, Z -8.0000, A 0.000, B 0.000, C 0.000 }
gfCNCPoint6[10807] = {X 522.7511, Y 50.1494, Z -8.0000, A 0.000, B 0.000, C 0.000 }
gfCNCPoint6[10808] = {X 522.0427, Y 50.5405, Z -8.0000, A 0.000, B 0.000, C 0.000 }
gfCNCPoint6[10809] = {X 521.2720, Y 50.7868, Z -8.0000, A 0.000, B 0.000, C 0.000 }
gfCNCPoint6[10810] = {X 520.4681, Y 50.8791, Z -8.0000, A 0.000, B 0.000, C 0.000 }
gfCNCPoint6[10811] = {X 519.7998, Y 50.8791, Z -8.0000, A 0.000, B 0.000, C 0.000 }
gfCNCPoint6[10812] = {X 518.9097, Y 50.7788, Z -8.0000, A 0.000, B 0.000, C 0.000 }
gfCNCPoint6[10813] = {X 518.0642, Y 50.4830, Z -8.0000, A 0.000, B 0.000, C 0.000 }
gfCNCPoint6[10814] = {X 517.3058, Y 50.0064, Z -8.0000, A 0.000, B 0.000, C 0.000 }
gfCNCPoint6[10815] = {X 516.6724, Y 49.3731, Z -8.0000, A 0.000, B 0.000, C 0.000 }
gfCNCPoint6[10816] = {X 516.1959, Y 48.6147, Z -8.0000, A 0.000, B 0.000, C 0.000 }
gfCNCPoint6[10817] = {X 515.9001, Y 47.7692, Z -8.0000, A 0.000, B 0.000, C 0.000 }
gfCNCPoint6[10818] = {X 515.7998, Y 46.8791, Z -8.0000, A 0.000, B 0.000, C 0.000 }
gfCNCPoint6[10819] = {X 515.7998, Y 39.9011, Z -8.0000, A 0.000, B 0.000, C 0.000 }
gfCNCPoint6[10820] = {X 515.9001, Y 39.0110, Z -8.0000, A 0.000, B 0.000, C 0.000 }
gfCNCPoint6[10821] = {X 516.1959, Y 38.1656, Z -8.0000, A 0.000, B 0.000, C 0.000 }
gfCNCPoint6[10822] = {X 516.6725, Y 37.4071, Z -8.0000, A 0.000, B 0.000, C 0.000 }
gfCNCPoint6[10823] = {X 517.3058, Y 36.7738, Z -8.0000, A 0.000, B 0.000, C 0.000 }
gfCNCPoint6[10824] = {X 518.0643, Y 36.2972, Z -8.0000, A 0.000, B 0.000, C 0.000 }
gfCNCPoint6[10825] = {X 518.9097, Y 36.0014, Z -8.0000, A 0.000, B 0.000, C 0.000 }
gfCNCPoint6[10826] = {X 519.7998, Y 35.9011, Z -8.0000, A 0.000, B 0.000, C 0.000 }
gfCNCPoint6[10827] = {X 520.5225, Y 35.9015, Z -8.0000, A 0.000, B 0.000, C 0.000 }
gfCNCPoint6[10828] = {X 521.3204, Y 35.9929, Z -8.0000, A 0.000, B 0.000, C 0.000 }
gfCNCPoint6[10829] = {X 522.0839, Y 36.2419, Z -8.0000, A 0.000, B 0.000, C 0.000 }
gfCNCPoint6[10830] = {X 522.7823, Y 36.6385, Z -8.0000, A 0.000, B 0.000, C 0.000 }
gfCNCPoint6[10831] = {X 523.3874, Y 37.1665, Z -8.0000, A 0.000, B 0.000, C 0.000 }
gfCNCPoint6[10832] = {X 523.8748, Y 37.8048, Z -8.0000, A 0.000, B 0.000, C 0.000 }
gfCNCPoint6[10833] = {X 534.9519, Y 37.8048, Z -8.0000, A 0.000, B 0.000, C 0.000 }
gfCNCPoint6[10834] = {X 534.9519, Y 33.6464, Z -8.0000, A 0.000, B 0.000, C 0.000 }
gfCNCPoint6[10835] = {X 529.9340, Y 33.6463, Z -8.0000, A 0.000, B 0.000, C 0.000 }
gfCNCPoint6[10836] = {X 529.8220, Y 33.8193, Z -8.0000, A 0.000, B 0.000, C 0.000 }
gfCNCPoint6[10837] = {X 529.1826, Y 34.5420, Z -8.0000, A 0.000, B 0.000, C 0.000 }
gfCNCPoint6[10838] = {X 528.3886, Y 35.0906, Z -8.0000, A 0.000, B 0.000, C 0.000 }
gfCNCPoint6[10839] = {X 527.4863, Y 35.4331, Z -8.0000, A 0.000, B 0.000, C 0.000 }
gfCNCPoint6[10840] = {X 526.5283, Y 35.5495, Z -8.0000, A 0.000, B 0.000, C 0.000 }
gfCNCPoint6[10841] = {X 525.8868, Y 35.5495, Z -8.0000, A 0.000, B 0.000, C 0.000 }
gfCNCPoint6[10842] = {X 524.9967, Y 35.4492, Z -8.0000, A 0.000, B 0.000, C 0.000 }
gfCNCPoint6[10843] = {X 524.1512, Y 35.1533, Z -8.0000, A 0.000, B 0.000, C 0.000 }
gfCNCPoint6[10844] = {X 523.3928, Y 34.6768, Z -8.0000, A 0.000, B 0.000, C 0.000 }
gfCNCPoint6[10845] = {X 522.7594, Y 34.0434, Z -8.0000, A 0.000, B 0.000, C 0.000 }
gfCNCPoint6[10846] = {X 522.2829, Y 33.2850, Z -8.0000, A 0.000, B 0.000, C 0.000 }
gfCNCPoint6[10847] = {X 521.9870, Y 32.4395, Z -8.0000, A 0.000, B 0.000, C 0.000 }
gfCNCPoint6[10848] = {X 521.8868, Y 31.5495, Z -8.0000, A 0.000, B 0.000, C 0.000 }
gfCNCPoint6[10849] = {X 521.8868, Y 24.5714, Z -8.0000, A 0.000, B 0.000, C 0.000 }
gfCNCPoint6[10850] = {X 521.9870, Y 23.6813, Z -8.0000, A 0.000, B 0.000, C 0.000 }
gfCNCPoint6[10851] = {X 522.2829, Y 22.8359, Z -8.0000, A 0.000, B 0.000, C 0.000 }
gfCNCPoint6[10852] = {X 522.7594, Y 22.0775, Z -8.0000, A 0.000, B 0.000, C 0.000 }
gfCNCPoint6[10853] = {X 523.3928, Y 21.4441, Z -8.0000, A 0.000, B 0.000, C 0.000 }
gfCNCPoint6[10854] = {X 524.1512, Y 20.9675, Z -8.0000, A 0.000, B 0.000, C 0.000 }
gfCNCPoint6[10855] = {X 524.9967, Y 20.6717, Z -8.0000, A 0.000, B 0.000, C 0.000 }
gfCNCPoint6[10856] = {X 525.8868, Y 20.5714, Z -8.0000, A 0.000, B 0.000, C 0.000 }
gfCNCPoint6[10857] = {X 526.5664, Y 20.5716, Z -8.0000, A 0.000, B 0.000, C 0.000 }
gfCNCPoint6[10858] = {X 527.3627, Y 20.6594, Z -8.0000, A 0.000, B 0.000, C 0.000 }
gfCNCPoint6[10859] = {X 528.1256, Y 20.9041, Z -8.0000, A 0.000, B 0.000, C 0.000 }
gfCNCPoint6[10860] = {X 528.8243, Y 21.2959, Z -8.0000, A 0.000, B 0.000, C 0.000 }
gfCNCPoint6[10861] = {X 529.4310, Y 21.8191, Z -8.0000, A 0.000, B 0.000, C 0.000 }
gfCNCPoint6[10862] = {X 529.9212, Y 22.4527, Z -8.0000, A 0.000, B 0.000, C 0.000 }
gfCNCPoint6[10863] = {X 534.9519, Y 22.4527, Z -8.0000, A 0.000, B 0.000, C 0.000 }
gfCNCPoint6[10864] = {X 534.9519, Y 19.3828, Z -8.0000, A 0.000, B 0.000, C 0.000 }
gfCNCPoint6[10865] = {X 524.0174, Y 19.3828, Z -8.0000, A 0.000, B 0.000, C 0.000 }
gfCNCPoint6[10866] = {X 523.9042, Y 19.5558, Z -8.0000, A 0.000, B 0.000, C 0.000 }
gfCNCPoint6[10867] = {X 523.2648, Y 20.2784, Z -8.0000, A 0.000, B 0.000, C 0.000 }
gfCNCPoint6[10868] = {X 522.4708, Y 20.8269, Z -8.0000, A 0.000, B 0.000, C 0.000 }
gfCNCPoint6[10869] = {X 521.5687, Y 21.1693, Z -8.0000, A 0.000, B 0.000, C 0.000 }
gfCNCPoint6[10870] = {X 520.6107, Y 21.2857, Z -8.0000, A 0.000, B 0.000, C 0.000 }
gfCNCPoint6[10871] = {X 519.9691, Y 21.2857, Z -8.0000, A 0.000, B 0.000, C 0.000 }
gfCNCPoint6[10872] = {X 519.0790, Y 21.1854, Z -8.0000, A 0.000, B 0.000, C 0.000 }
gfCNCPoint6[10873] = {X 518.2336, Y 20.8896, Z -8.0000, A 0.000, B 0.000, C 0.000 }
gfCNCPoint6[10874] = {X 517.4751, Y 20.4130, Z -8.0000, A 0.000, B 0.000, C 0.000 }
